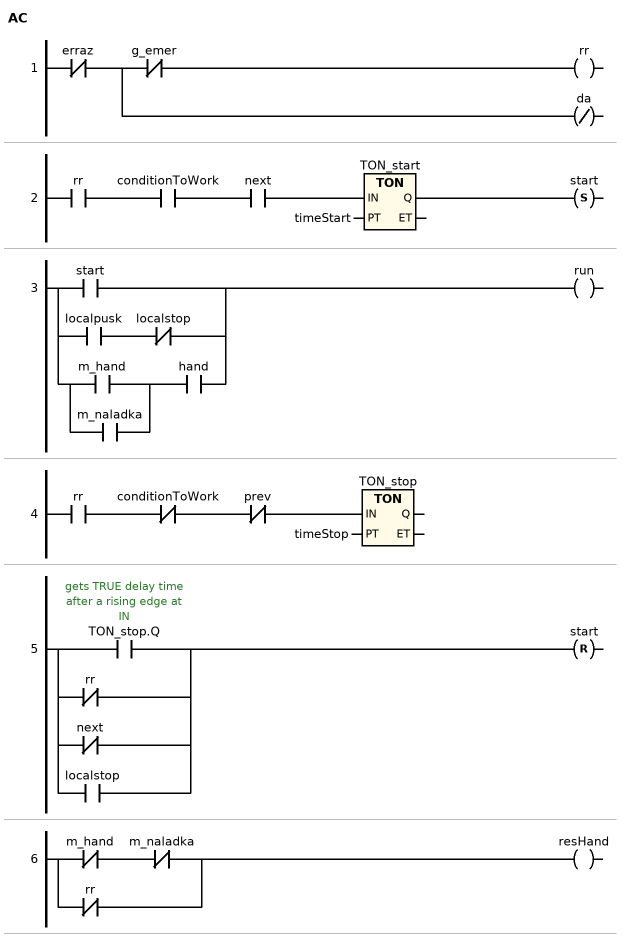
// NETWORK 1
_w1 := NOT erraz;
rr := _w1 AND NOT g_emer;
da := NOT _w1;

// NETWORK 2
TON_start(IN := rr AND conditionToWork AND next, PT := timeStart); // TON
start S= TON_start.Q;

// NETWORK 3
run := start OR localpusk AND NOT localstop OR (m_hand OR m_naladka) AND hand;

// NETWORK 4
TON_stop(IN := rr AND NOT conditionToWork AND NOT prev, PT := timeStop); // TON

// NETWORK 5
//   TON_stop.Q: gets TRUE delay time after a rising edge at IN
start R= TON_stop.Q OR NOT rr OR NOT next OR localstop;

// NETWORK 6
resHand := NOT m_hand AND NOT m_naladka OR NOT rr;

END_FUNCTION_BLOCK

// PLC_241/Application/FB/Noria/N
FUNCTION_BLOCK N
VAR_INPUT
	dks: BOOL;
	dsl1: BOOL;
	dsl2: BOOL;
	dp: BOOL;
	localpusk: BOOL;
	localstop: BOOL;
	erraz: BOOL;
	timeDKS: TIME;
	timeDSL: TIME;
	timeDP: TIME;
	timeStart: TIME;
	timeStop: TIME;
	next: BOOL;
	prev: BOOL;
	conditionToWork: BOOL;
	ressetErrors: BOOL;
	g_emer: BOOL;
	m_hand: BOOL;
	m_naladka: BOOL;
	hand: BOOL;
	offdks: BOOL;
	offdsl1: BOOL;
	offdsl2: BOOL;
	offdp: BOOL;
END_VAR
VAR_OUTPUT
	run: BOOL;
	rr: BOOL;
	da: BOOL;
	errDKS: BOOL;
	errDSL1: BOOL;
	errDSL2: BOOL;
	errDP: BOOL;
	resHand: BOOL;
END_VAR
VAR
	TON_DKS1: TON;
	TON_DKS2: TON;
	TON_DSL1: TON;
	TON_DSL2: TON;
	TON_DP: TON;
	TON_start: TON;
	start: BOOL;
	TON_stop: TON;
END_VAR
VAR // added by the converter: edge detectors and wires of the graphical bodies
    _w1 : BOOL;
END_VAR

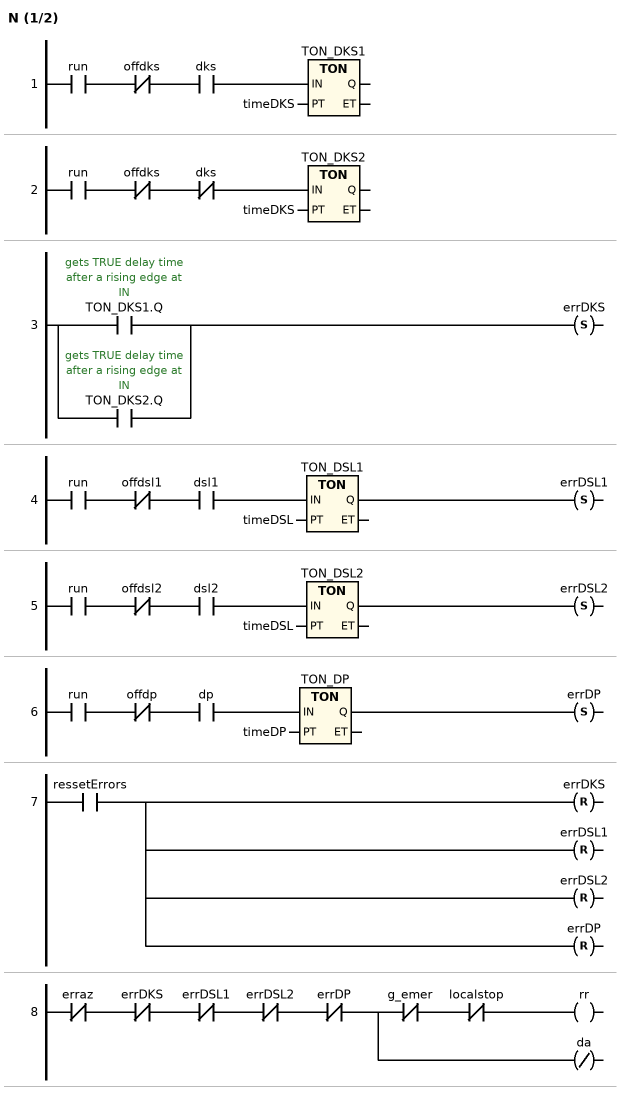
// NETWORK 1
TON_DKS1(IN := run AND NOT offdks AND dks, PT := timeDKS); // TON

// NETWORK 2
TON_DKS2(IN := run AND NOT offdks AND NOT dks, PT := timeDKS); // TON

// NETWORK 3
//   TON_DKS1.Q: gets TRUE delay time after a rising edge at IN
//   TON_DKS2.Q: gets TRUE delay time after a rising edge at IN
errDKS S= TON_DKS1.Q OR TON_DKS2.Q;

// NETWORK 4
TON_DSL1(IN := run AND NOT offdsl1 AND dsl1, PT := timeDSL); // TON
errDSL1 S= TON_DSL1.Q;

// NETWORK 5
TON_DSL2(IN := run AND NOT offdsl2 AND dsl2, PT := timeDSL); // TON
errDSL2 S= TON_DSL2.Q;

// NETWORK 6
TON_DP(IN := run AND NOT offdp AND dp, PT := timeDP); // TON
errDP S= TON_DP.Q;

// NETWORK 7
errDKS R= ressetErrors;
errDSL1 R= ressetErrors;
errDSL2 R= ressetErrors;
errDP R= ressetErrors;

// NETWORK 8
_w1 := NOT erraz AND NOT errDKS AND NOT errDSL1 AND NOT errDSL2 AND NOT errDP;
rr := _w1 AND NOT g_emer AND NOT localstop;
da := NOT _w1;

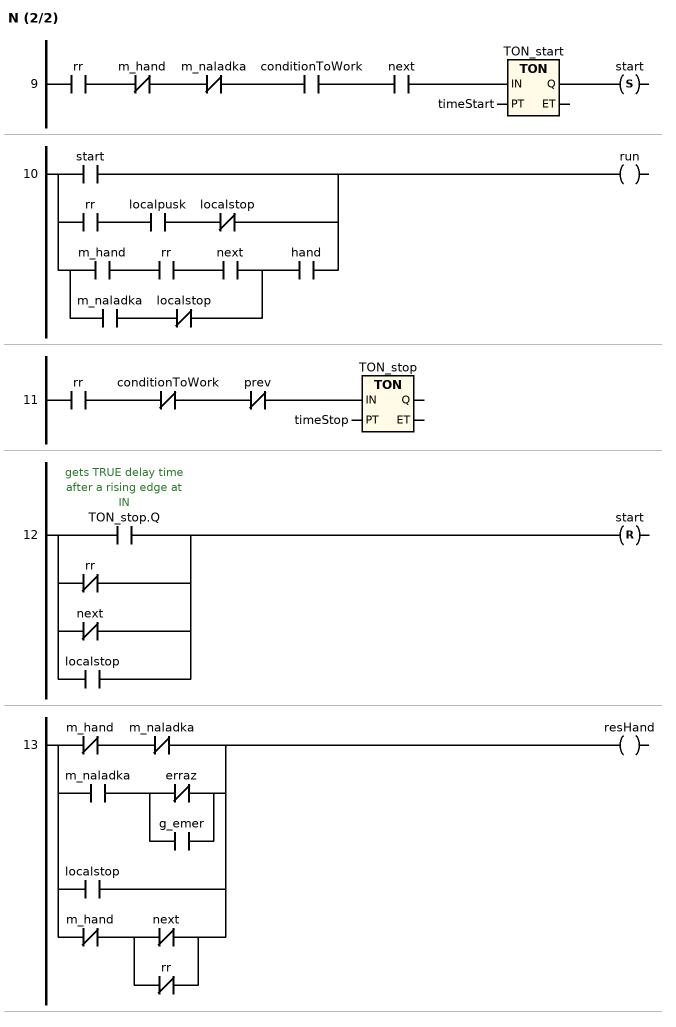
// NETWORK 9
TON_start(IN := rr AND NOT m_hand AND NOT m_naladka AND conditionToWork AND next, PT := timeStart); // TON
start S= TON_start.Q;

// NETWORK 10
run := start OR rr AND localpusk AND NOT localstop OR (m_hand AND rr AND next OR m_naladka AND NOT localstop) AND hand;

// NETWORK 11
TON_stop(IN := rr AND NOT conditionToWork AND NOT prev, PT := timeStop); // TON

// NETWORK 12
//   TON_stop.Q: gets TRUE delay time after a rising edge at IN
start R= TON_stop.Q OR NOT rr OR NOT next OR localstop;

// NETWORK 13
resHand := NOT m_hand AND NOT m_naladka OR m_naladka AND (NOT erraz OR g_emer) OR localstop OR NOT m_hand AND (NOT next OR NOT rr);

END_FUNCTION_BLOCK

// PLC_241/Application/FB/Flap/KP
FUNCTION_BLOCK KP
VAR_INPUT
	erraz: BOOL;
	pol_1: BOOL;
	pol_2: BOOL;
	conditionToWork_pol_1: BOOL;
	conditionToWork_pol_2: BOOL;
	timeLT: TIME;
	timePol_1: TIME;
	timePol_2: TIME;
	ressetErrors: BOOL;
	g_emer: BOOL;
	m_hand: BOOL;
	m_naladka: BOOL;
	hand_pol_1: BOOL;
	hand_pol_2: BOOL;
END_VAR
VAR_OUTPUT
	runPol_1: BOOL;
	runPol_2: BOOL;
	rr: BOOL;
	da: BOOL;
	errLT: BOOL;
	errConc: BOOL;
	stPol_1: BOOL;
	stPol_2: BOOL;
	resHand_pol_1: BOOL;
	resHand_pol_2: BOOL;
END_VAR
VAR
	TON_POL_1: TON;
	TON_LT: TON;
	TON_POL_2: TON;
END_VAR
VAR // added by the converter: edge detectors and wires of the graphical bodies
    _w1, _w2 : BOOL;
END_VAR

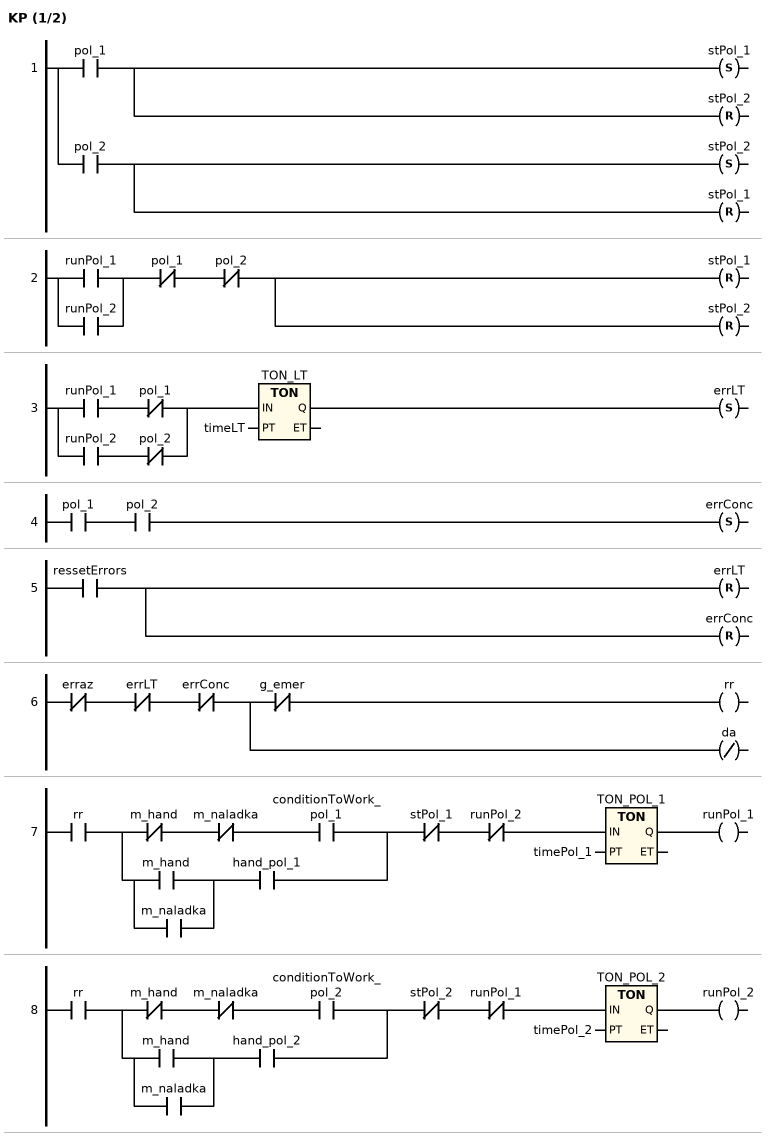
// NETWORK 1
stPol_1 S= pol_1;
stPol_2 R= pol_1;
stPol_2 S= pol_2;
stPol_1 R= pol_2;

// NETWORK 2
_w1 := (runPol_1 OR runPol_2) AND NOT pol_1 AND NOT pol_2;
stPol_1 R= _w1;
stPol_2 R= _w1;

// NETWORK 3
TON_LT(IN := runPol_1 AND NOT pol_1 OR runPol_2 AND NOT pol_2, PT := timeLT); // TON
errLT S= TON_LT.Q;

// NETWORK 4
errConc S= pol_1 AND pol_2;

// NETWORK 5
errLT R= ressetErrors;
errConc R= ressetErrors;

// NETWORK 6
_w2 := NOT erraz AND NOT errLT AND NOT errConc;
rr := _w2 AND NOT g_emer;
da := NOT _w2;

// NETWORK 7
TON_POL_1(IN := rr AND (NOT m_hand AND NOT m_naladka AND conditionToWork_pol_1 OR (m_hand OR m_naladka) AND hand_pol_1) AND NOT stPol_1 AND NOT runPol_2, PT := timePol_1); // TON
runPol_1 := TON_POL_1.Q;

// NETWORK 8
TON_POL_2(IN := rr AND (NOT m_hand AND NOT m_naladka AND conditionToWork_pol_2 OR (m_hand OR m_naladka) AND hand_pol_2) AND NOT stPol_2 AND NOT runPol_1, PT := timePol_2); // TON
runPol_2 := TON_POL_2.Q;

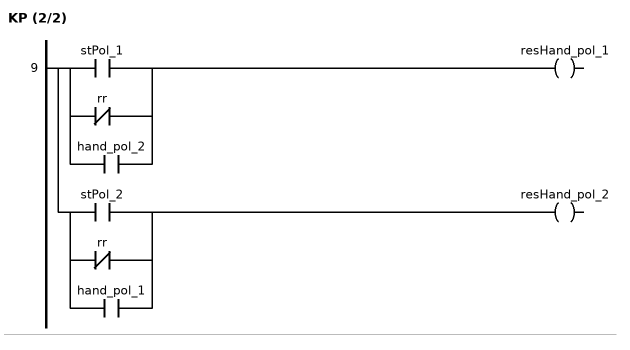
// NETWORK 9
resHand_pol_1 := stPol_1 OR NOT rr OR hand_pol_2;
resHand_pol_2 := stPol_2 OR NOT rr OR hand_pol_1;

END_FUNCTION_BLOCK

// PLC_241/Application/FB/scalperator/SCLP
FUNCTION_BLOCK SCLP
VAR_INPUT
	errpch: BOOL;
	prev: BOOL;
	next: BOOL;
	conditionToWork: BOOL;
	timeStart: TIME;
	timeStop: TIME;
	ressetErrors: BOOL;
	g_emer: BOOL;
	m_hand: BOOL;
	m_naladka: BOOL;
	hand: BOOL;
	
END_VAR
VAR_OUTPUT
	runPuskatel: BOOL;
	runPCH: BOOL;
	runRessetPCH: BOOL;
	rr: BOOL;
	da: BOOL;
	resHand: BOOL;
END_VAR
VAR
	TON_Start: TON;
	start: BOOL;
	TON_Stop: TON;
	TON_PCH_ON: TON;
END_VAR
VAR // added by the converter: edge detectors and wires of the graphical bodies
    _w1 : BOOL;
END_VAR

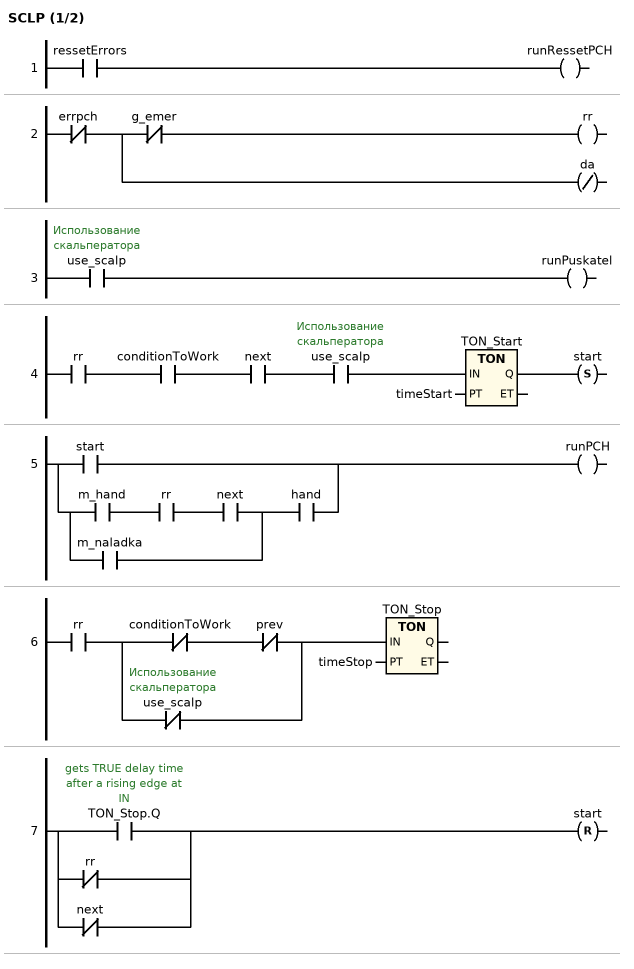
// NETWORK 1
runRessetPCH := ressetErrors;

// NETWORK 2
_w1 := NOT errpch;
rr := _w1 AND NOT g_emer;
da := NOT _w1;

// NETWORK 3
//   use_scalp: Использование скальператора
runPuskatel := use_scalp;

// NETWORK 4
//   use_scalp: Использование скальператора
TON_Start(IN := rr AND conditionToWork AND next AND use_scalp, PT := timeStart); // TON
start S= TON_Start.Q;

// NETWORK 5
runPCH := start OR (m_hand AND rr AND next OR m_naladka) AND hand;

// NETWORK 6
//   use_scalp: Использование скальператора
TON_Stop(IN := rr AND (NOT conditionToWork AND NOT prev OR NOT use_scalp), PT := timeStop); // TON

// NETWORK 7
//   TON_Stop.Q: gets TRUE delay time after a rising edge at IN
start R= TON_Stop.Q OR NOT rr OR NOT next;

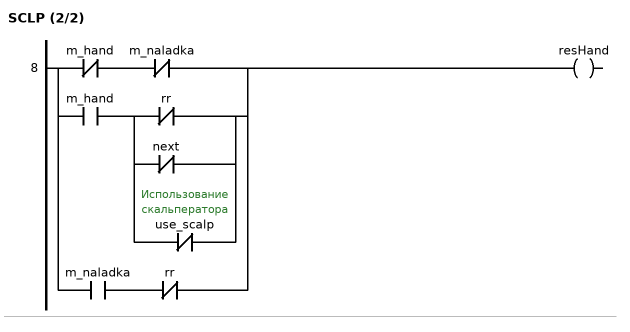
// NETWORK 8
//   use_scalp: Использование скальператора
resHand := NOT m_hand AND NOT m_naladka OR m_hand AND (NOT rr OR NOT next OR NOT use_scalp) OR m_naladka AND NOT rr;

END_FUNCTION_BLOCK

// PLC_241/Application/FB/SH/Z
FUNCTION_BLOCK Z
VAR_INPUT
	erraz: BOOL;
	opened: BOOL;
	closed: BOOL;
	next: BOOL;
	prev: BOOL;
	conditionToWork: BOOL;
	timeLT: TIME;
	timeOpen: TIME;
	timeClose: TIME;
	g_emer: BOOL;
	ressetErrors: BOOL;
	m_hand: BOOL;
	m_naladka: BOOL;
	hand_open: BOOL;
	hand_close: BOOL;
END_VAR
VAR_OUTPUT
	runOpen: BOOL; 
	runClose: BOOL;
	rr: BOOL;
	da: BOOL;
	errLT: BOOL;
	errConc: BOOL;
	resHand_open: BOOL;
	resHand_close: BOOL;
END_VAR
VAR
	TON_LT: TON;
	TON_open: TON;
	TON_close: TON;
END_VAR
VAR // added by the converter: edge detectors and wires of the graphical bodies
    _w1 : BOOL;
END_VAR

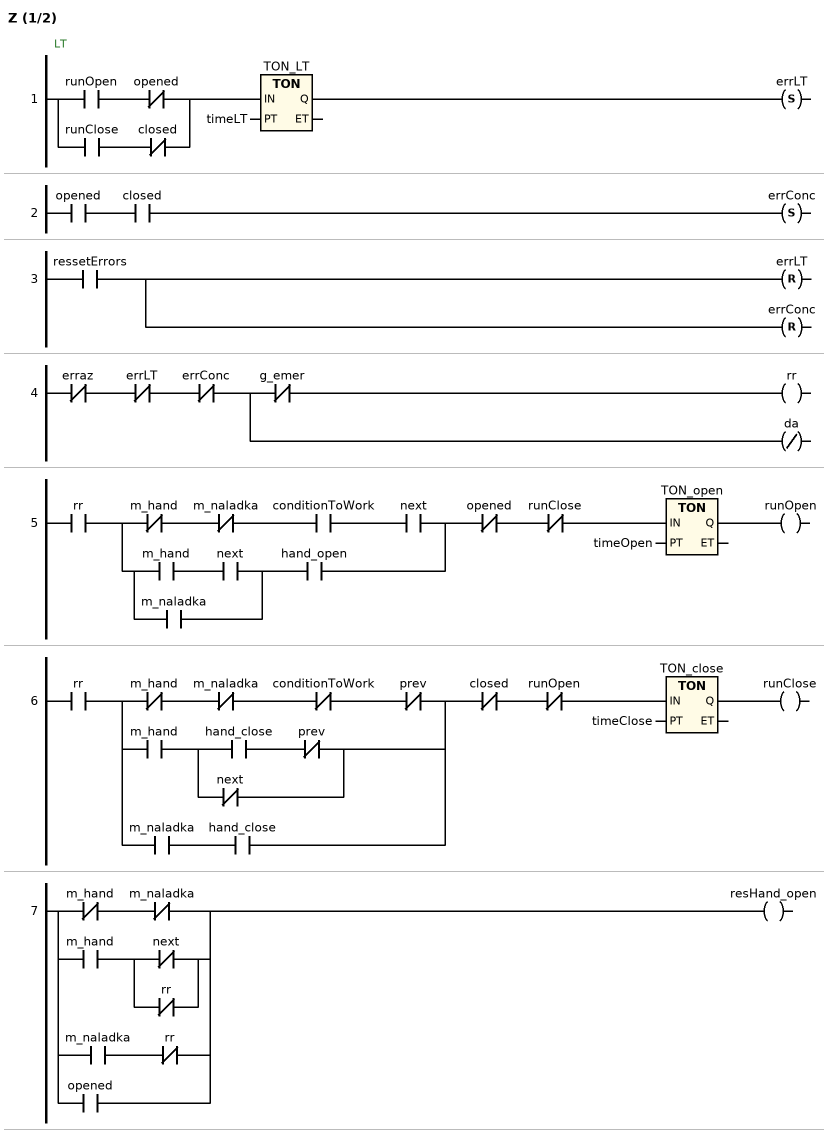
// NETWORK 1
// LT
TON_LT(IN := runOpen AND NOT opened OR runClose AND NOT closed, PT := timeLT); // TON
errLT S= TON_LT.Q;

// NETWORK 2
errConc S= opened AND closed;

// NETWORK 3
errLT R= ressetErrors;
errConc R= ressetErrors;

// NETWORK 4
_w1 := NOT erraz AND NOT errLT AND NOT errConc;
rr := _w1 AND NOT g_emer;
da := NOT _w1;

// NETWORK 5
TON_open(IN := rr AND (NOT m_hand AND NOT m_naladka AND conditionToWork AND next OR (m_hand AND next OR m_naladka) AND hand_open) AND NOT opened AND NOT runClose, PT := timeOpen); // TON
runOpen := TON_open.Q;

// NETWORK 6
TON_close(IN := rr AND (NOT m_hand AND NOT m_naladka AND NOT conditionToWork AND NOT prev OR m_hand AND (hand_close AND NOT prev OR NOT next) OR m_naladka AND hand_close) AND NOT closed AND NOT runOpen, PT := timeClose); // TON
runClose := TON_close.Q;

// NETWORK 7
resHand_open := NOT m_hand AND NOT m_naladka OR m_hand AND (NOT next OR NOT rr) OR m_naladka AND NOT rr OR opened;

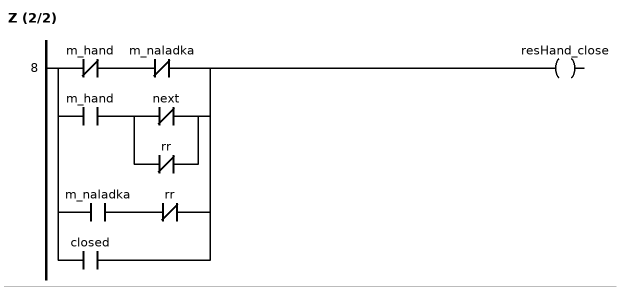
// NETWORK 8
resHand_close := NOT m_hand AND NOT m_naladka OR m_hand AND (NOT next OR NOT rr) OR m_naladka AND NOT rr OR closed;

END_FUNCTION_BLOCK

// PLC_241/Application/POU/prgLoad_K
PROGRAM prgLoad_K
VAR
	N_21200: N;
	Step_K: INT;
	imp_K: BOOL;
	imp_dvy_201: BOOL;
	imp_dvy_202: BOOL;
	imp_dvy_203: BOOL;
	imp_dvy_204: BOOL;
	TON_imp_bunk_201: TON;
	pause_load_K: BOOL;
	TON_imp_bunk_202: TON;
	TON_imp_bunk_203: TON;
	TON_imp_bunk_204: TON;
	TON_pause_K: TON;
	Shnek_21300: Shnek;
	TOF_next_shnek_21300: TOF;
	TP_STEP_K: TP;
	Z_21310: Z;
	Z_21320: Z;
	Z_21330: Z;
	check_K: BOOL;
	imp_nextBunk_K: BOOL;
	TON_Resset_modeLoad_k: TON;
END_VAR
VAR // added by the converter: edge detectors and wires of the graphical bodies
    _rt1, _rt2, _rt3, _rt4, _rt5, _rt6, _rt7, _rt8, _rt9, _rt10, _rt11, _rt12, _rt13 : R_TRIG;
    _w1, _w2, _w3, _w4, _w5, _w6 : BOOL;
END_VAR

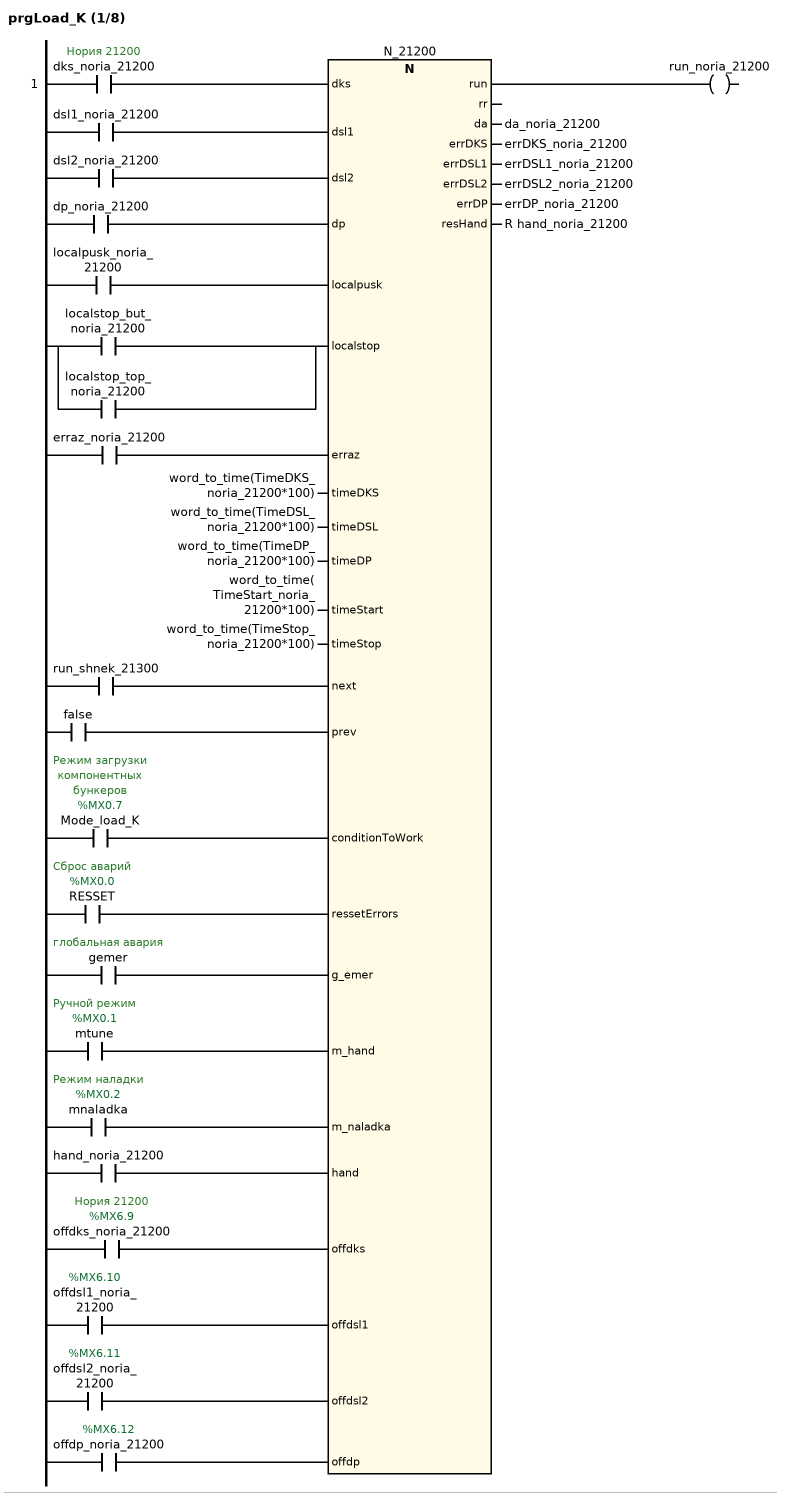
// NETWORK 1
//   dks_noria_21200: Нория 21200
//   Mode_load_K: Режим загрузки компонентных бункеров | AT %MX0.7
//   RESSET: Сброс аварий | AT %MX0.0
//   gemer: глобальная авария
//   mtune: Ручной режим | AT %MX0.1
//   mnaladka: Режим наладки | AT %MX0.2
//   offdks_noria_21200: Нория 21200 | AT %MX6.9
//   offdsl1_noria_21200: AT %MX6.10
//   offdsl2_noria_21200: AT %MX6.11
//   offdp_noria_21200: AT %MX6.12
//   errDKS_noria_21200: Нория 21200
N_21200(
    dks := dks_noria_21200,
    dsl1 := dsl1_noria_21200,
    dsl2 := dsl2_noria_21200,
    dp := dp_noria_21200,
    localpusk := localpusk_noria_21200,
    localstop := localstop_but_noria_21200 OR localstop_top_noria_21200,
    erraz := erraz_noria_21200,
    timeDKS := word_to_time(TimeDKS_noria_21200*100),
    timeDSL := word_to_time(TimeDSL_noria_21200*100),
    timeDP := word_to_time(TimeDP_noria_21200*100),
    timeStart := word_to_time(TimeStart_noria_21200*100),
    timeStop := word_to_time(TimeStop_noria_21200*100),
    next := run_shnek_21300,
    prev := false,
    conditionToWork := Mode_load_K,
    ressetErrors := RESSET,
    g_emer := gemer,
    m_hand := mtune,
    m_naladka := mnaladka,
    hand := hand_noria_21200,
    offdks := offdks_noria_21200,
    offdsl1 := offdsl1_noria_21200,
    offdsl2 := offdsl2_noria_21200,
    offdp := offdp_noria_21200,
    da => da_noria_21200,
    errDKS => errDKS_noria_21200,
    errDSL1 => errDSL1_noria_21200,
    errDSL2 => errDSL2_noria_21200,
    errDP => errDP_noria_21200); // N
hand_noria_21200 R= N_21200.resHand;
run_noria_21200 := N_21200.run;

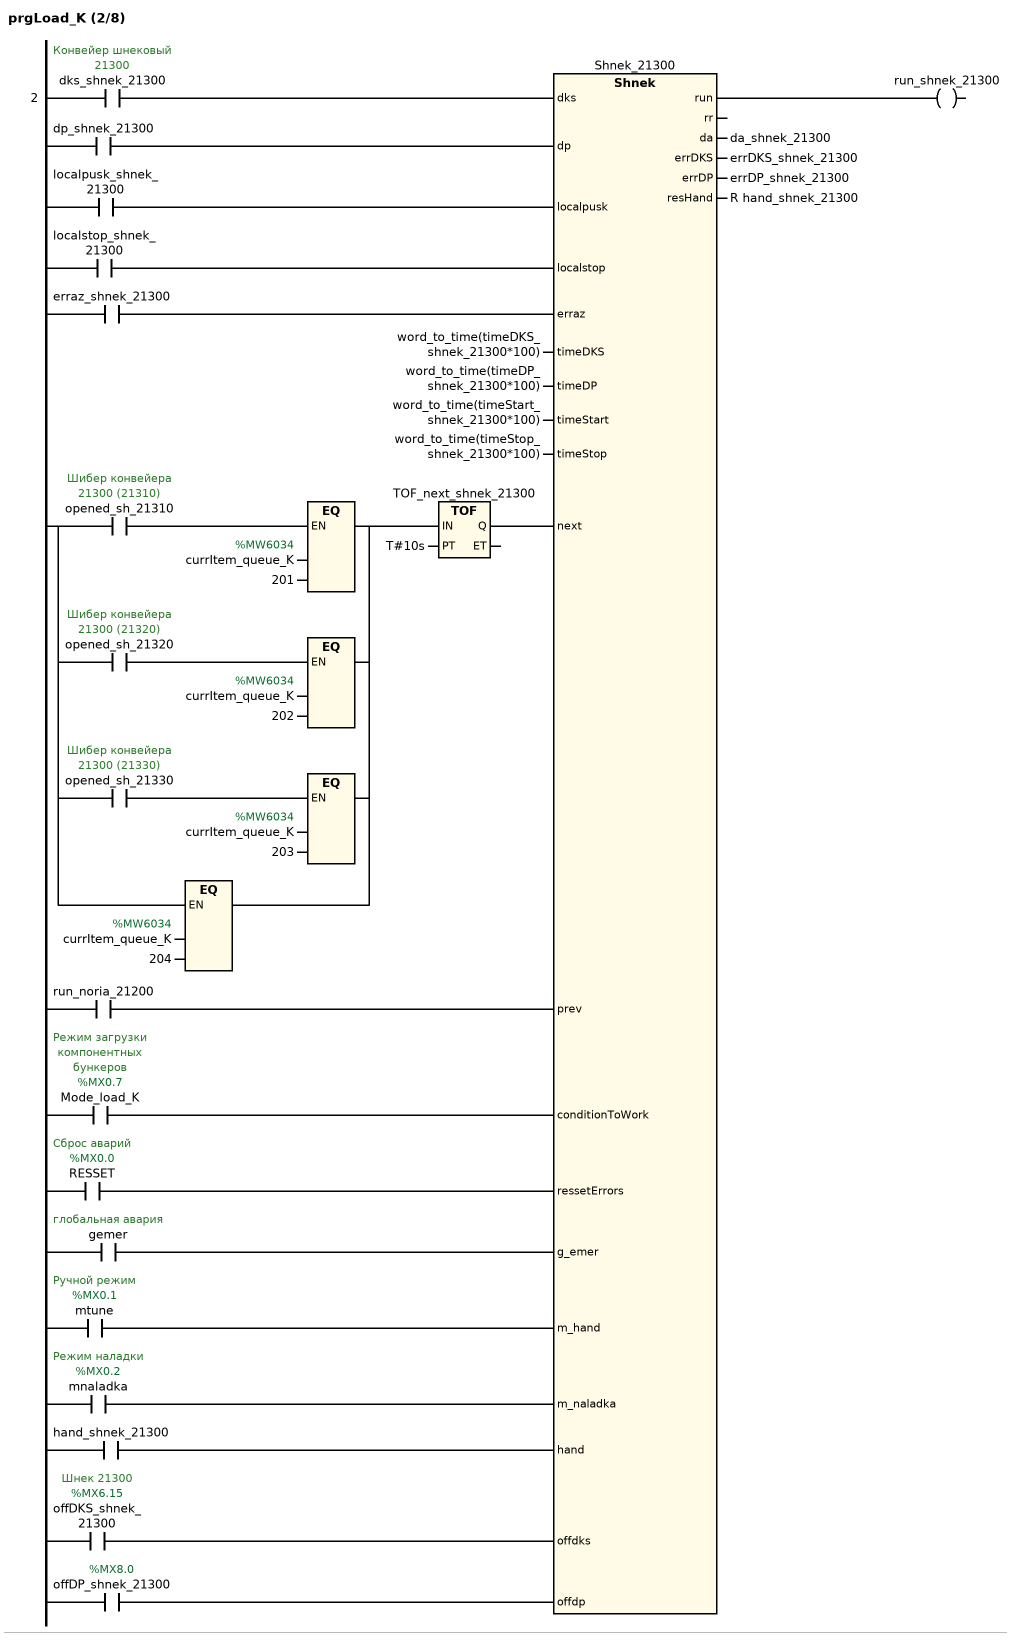
// NETWORK 2
//   dks_shnek_21300: Конвейер шнековый 21300
//   opened_sh_21310: Шибер конвейера 21300 (21310)
//   currItem_queue_K: Текущий бункер для загрузки в очереди компонентов | AT %MW6034
//   opened_sh_21320: Шибер конвейера 21300 (21320)
//   opened_sh_21330: Шибер конвейера 21300 (21330)
//   Mode_load_K: Режим загрузки компонентных бункеров | AT %MX0.7
//   RESSET: Сброс аварий | AT %MX0.0
//   gemer: глобальная авария
//   mtune: Ручной режим | AT %MX0.1
//   mnaladka: Режим наладки | AT %MX0.2
//   offDKS_shnek_21300: Шнек 21300 | AT %MX6.15
//   offDP_shnek_21300: AT %MX8.0
//   errDKS_shnek_21300: Шнек 21300
TOF_next_shnek_21300(IN := opened_sh_21310 AND currItem_queue_K = 201 OR opened_sh_21320 AND currItem_queue_K = 202 OR opened_sh_21330 AND currItem_queue_K = 203 OR currItem_queue_K = 204, PT := T#10s); // TOF
Shnek_21300(
    dks := dks_shnek_21300,
    dp := dp_shnek_21300,
    localpusk := localpusk_shnek_21300,
    localstop := localstop_shnek_21300,
    erraz := erraz_shnek_21300,
    timeDKS := word_to_time(timeDKS_shnek_21300*100),
    timeDP := word_to_time(timeDP_shnek_21300*100),
    timeStart := word_to_time(timeStart_shnek_21300*100),
    timeStop := word_to_time(timeStop_shnek_21300*100),
    next := TOF_next_shnek_21300.Q,
    prev := run_noria_21200,
    conditionToWork := Mode_load_K,
    ressetErrors := RESSET,
    g_emer := gemer,
    m_hand := mtune,
    m_naladka := mnaladka,
    hand := hand_shnek_21300,
    offdks := offDKS_shnek_21300,
    offdp := offDP_shnek_21300,
    da => da_shnek_21300,
    errDKS => errDKS_shnek_21300,
    errDP => errDP_shnek_21300); // Shnek
hand_shnek_21300 R= Shnek_21300.resHand;
run_shnek_21300 := Shnek_21300.run;

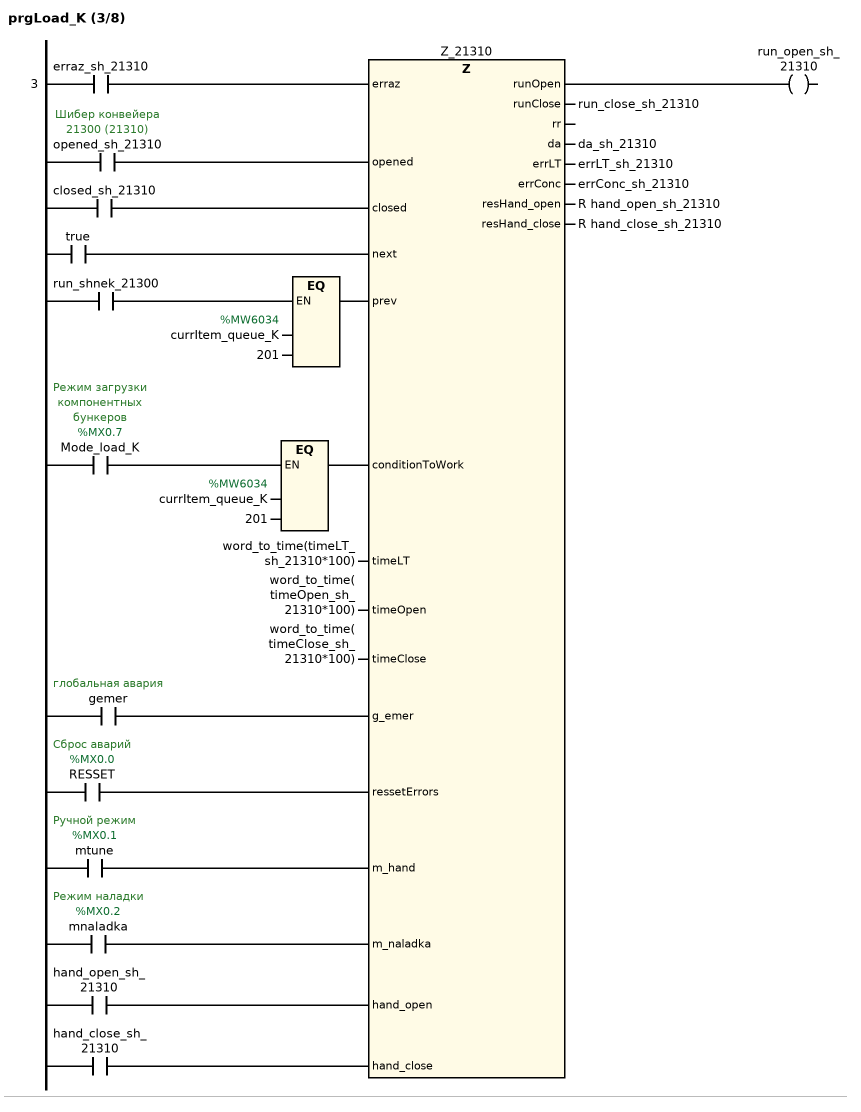
// NETWORK 3
//   opened_sh_21310: Шибер конвейера 21300 (21310)
//   currItem_queue_K: Текущий бункер для загрузки в очереди компонентов | AT %MW6034
//   Mode_load_K: Режим загрузки компонентных бункеров | AT %MX0.7
//   gemer: глобальная авария
//   RESSET: Сброс аварий | AT %MX0.0
//   mtune: Ручной режим | AT %MX0.1
//   mnaladka: Режим наладки | AT %MX0.2
//   errLT_sh_21310: Шибер 21310
Z_21310(
    erraz := erraz_sh_21310,
    opened := opened_sh_21310,
    closed := closed_sh_21310,
    next := true,
    prev := run_shnek_21300 AND currItem_queue_K = 201,
    conditionToWork := Mode_load_K AND currItem_queue_K = 201,
    timeLT := word_to_time(timeLT_sh_21310*100),
    timeOpen := word_to_time(timeOpen_sh_21310*100),
    timeClose := word_to_time(timeClose_sh_21310*100),
    g_emer := gemer,
    ressetErrors := RESSET,
    m_hand := mtune,
    m_naladka := mnaladka,
    hand_open := hand_open_sh_21310,
    hand_close := hand_close_sh_21310,
    runClose => run_close_sh_21310,
    da => da_sh_21310,
    errLT => errLT_sh_21310,
    errConc => errConc_sh_21310); // Z
hand_open_sh_21310 R= Z_21310.resHand_open;
hand_close_sh_21310 R= Z_21310.resHand_close;
run_open_sh_21310 := Z_21310.runOpen;

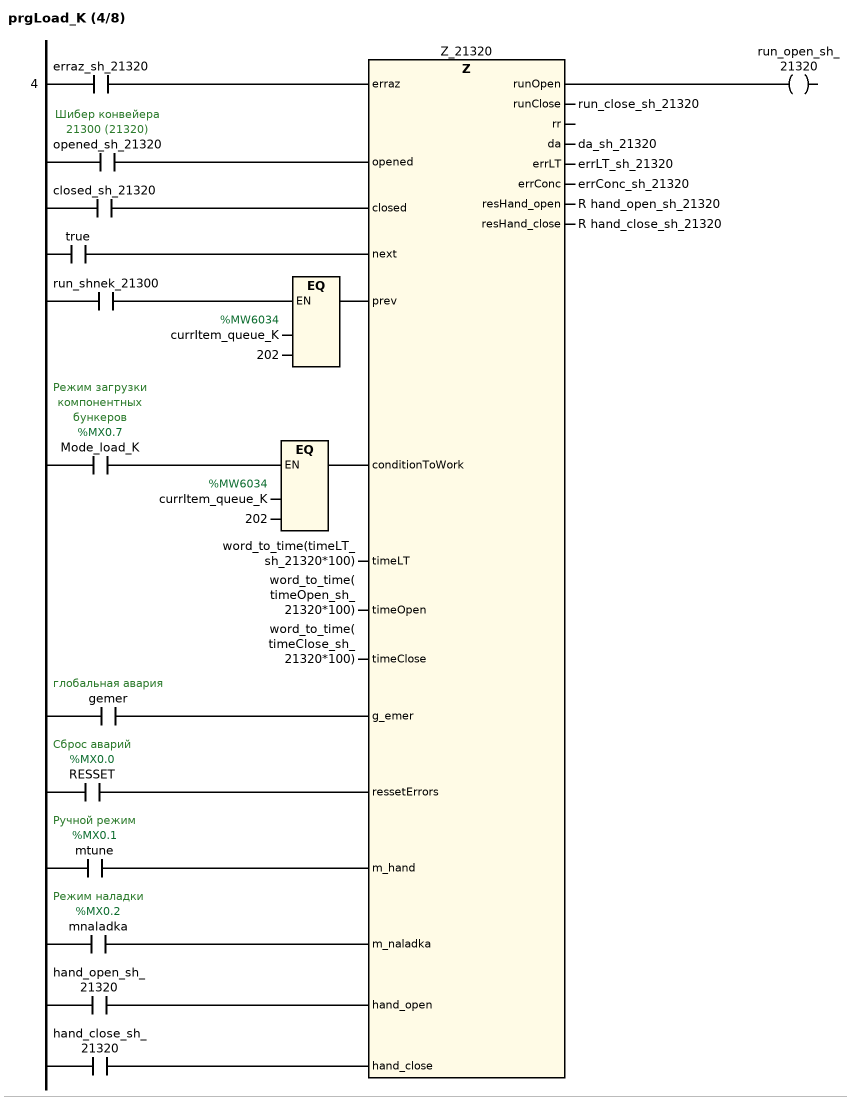
// NETWORK 4
//   opened_sh_21320: Шибер конвейера 21300 (21320)
//   currItem_queue_K: Текущий бункер для загрузки в очереди компонентов | AT %MW6034
//   Mode_load_K: Режим загрузки компонентных бункеров | AT %MX0.7
//   gemer: глобальная авария
//   RESSET: Сброс аварий | AT %MX0.0
//   mtune: Ручной режим | AT %MX0.1
//   mnaladka: Режим наладки | AT %MX0.2
//   errLT_sh_21320: Шибер 21320
Z_21320(
    erraz := erraz_sh_21320,
    opened := opened_sh_21320,
    closed := closed_sh_21320,
    next := true,
    prev := run_shnek_21300 AND currItem_queue_K = 202,
    conditionToWork := Mode_load_K AND currItem_queue_K = 202,
    timeLT := word_to_time(timeLT_sh_21320*100),
    timeOpen := word_to_time(timeOpen_sh_21320*100),
    timeClose := word_to_time(timeClose_sh_21320*100),
    g_emer := gemer,
    ressetErrors := RESSET,
    m_hand := mtune,
    m_naladka := mnaladka,
    hand_open := hand_open_sh_21320,
    hand_close := hand_close_sh_21320,
    runClose => run_close_sh_21320,
    da => da_sh_21320,
    errLT => errLT_sh_21320,
    errConc => errConc_sh_21320); // Z
hand_open_sh_21320 R= Z_21320.resHand_open;
hand_close_sh_21320 R= Z_21320.resHand_close;
run_open_sh_21320 := Z_21320.runOpen;

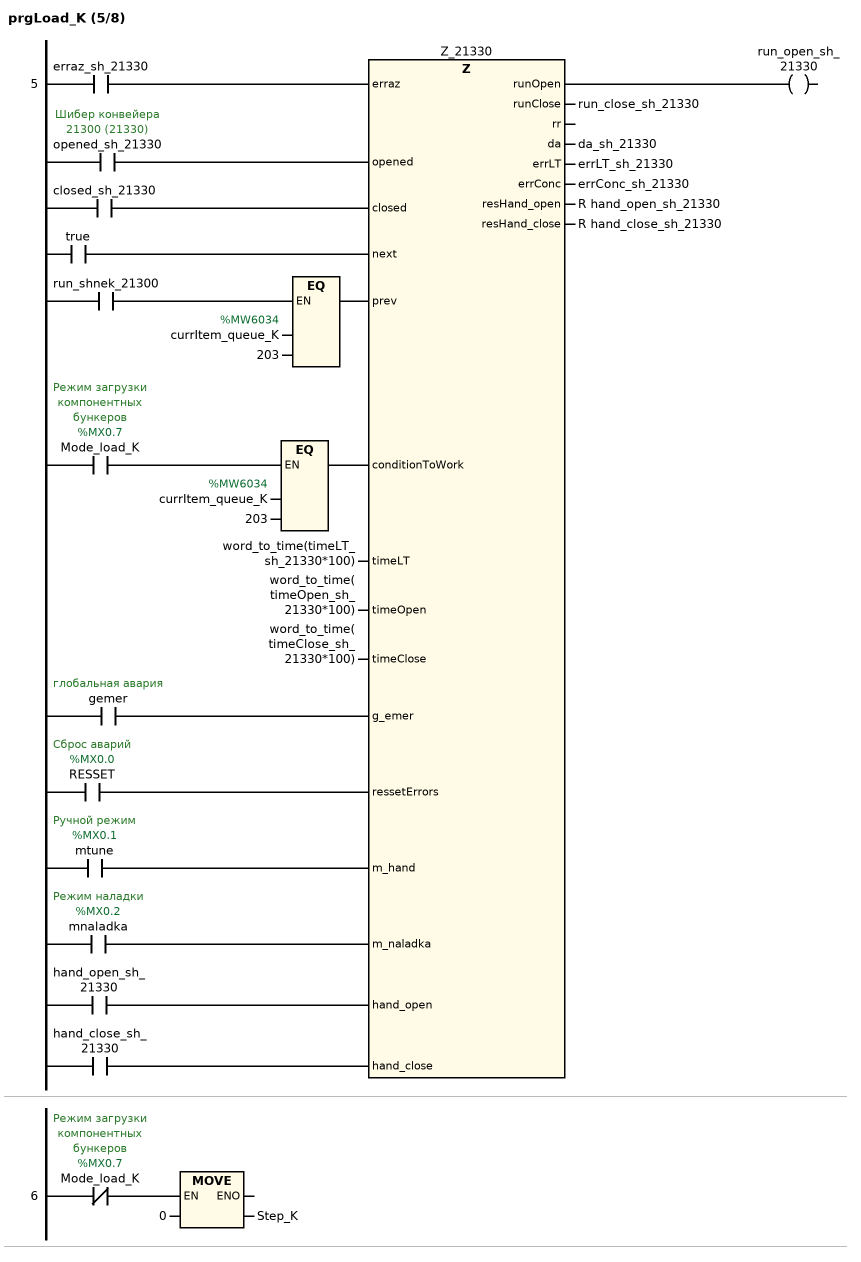
// NETWORK 5
//   opened_sh_21330: Шибер конвейера 21300 (21330)
//   currItem_queue_K: Текущий бункер для загрузки в очереди компонентов | AT %MW6034
//   Mode_load_K: Режим загрузки компонентных бункеров | AT %MX0.7
//   gemer: глобальная авария
//   RESSET: Сброс аварий | AT %MX0.0
//   mtune: Ручной режим | AT %MX0.1
//   mnaladka: Режим наладки | AT %MX0.2
//   errLT_sh_21330: Шибер 21330
Z_21330(
    erraz := erraz_sh_21330,
    opened := opened_sh_21330,
    closed := closed_sh_21330,
    next := true,
    prev := run_shnek_21300 AND currItem_queue_K = 203,
    conditionToWork := Mode_load_K AND currItem_queue_K = 203,
    timeLT := word_to_time(timeLT_sh_21330*100),
    timeOpen := word_to_time(timeOpen_sh_21330*100),
    timeClose := word_to_time(timeClose_sh_21330*100),
    g_emer := gemer,
    ressetErrors := RESSET,
    m_hand := mtune,
    m_naladka := mnaladka,
    hand_open := hand_open_sh_21330,
    hand_close := hand_close_sh_21330,
    runClose => run_close_sh_21330,
    da => da_sh_21330,
    errLT => errLT_sh_21330,
    errConc => errConc_sh_21330); // Z
hand_open_sh_21330 R= Z_21330.resHand_open;
hand_close_sh_21330 R= Z_21330.resHand_close;
run_open_sh_21330 := Z_21330.runOpen;

// NETWORK 6
//   Mode_load_K: Режим загрузки компонентных бункеров | AT %MX0.7
IF NOT Mode_load_K THEN Step_K := 0; END_IF

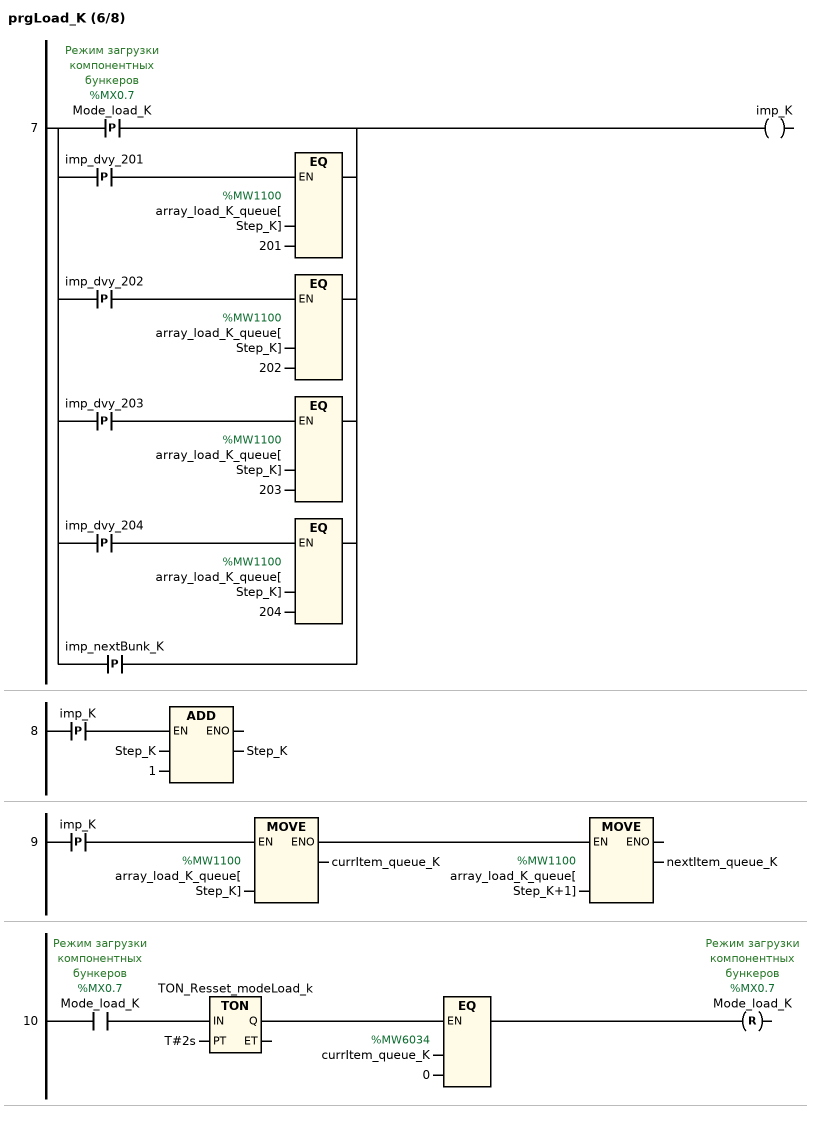
// NETWORK 7
//   Mode_load_K: Режим загрузки компонентных бункеров | AT %MX0.7
//   array_load_K_queue[Step_K]: Массив очереди загрузки компонентов | AT %MW1100
_rt1(CLK := Mode_load_K);
_rt2(CLK := imp_dvy_201);
_rt3(CLK := imp_dvy_202);
_rt4(CLK := imp_dvy_203);
_rt5(CLK := imp_dvy_204);
_rt6(CLK := imp_nextBunk_K);
imp_K := _rt1.Q OR _rt2.Q AND array_load_K_queue[Step_K] = 201 OR _rt3.Q AND array_load_K_queue[Step_K] = 202 OR _rt4.Q AND array_load_K_queue[Step_K] = 203 OR _rt5.Q AND array_load_K_queue[Step_K] = 204 OR _rt6.Q;

// NETWORK 8
_rt7(CLK := imp_K);
IF _rt7.Q THEN Step_K := Step_K + 1; END_IF

// NETWORK 9
//   array_load_K_queue[Step_K]: Массив очереди загрузки компонентов | AT %MW1100
//   currItem_queue_K: Текущий бункер для загрузки в очереди компонентов | AT %MW6034
//   array_load_K_queue[Step_K+1]: Массив очереди загрузки компонентов | AT %MW1100
//   nextItem_queue_K: Следующий бункер для загрузки в очереди компонентов | AT %MW6035
_rt8(CLK := imp_K);
_w1 := _rt8.Q;
IF _w1 THEN currItem_queue_K := array_load_K_queue[Step_K]; END_IF
IF _w1 THEN nextItem_queue_K := array_load_K_queue[Step_K+1]; END_IF

// NETWORK 10
//   Mode_load_K: Режим загрузки компонентных бункеров | AT %MX0.7
//   currItem_queue_K: Текущий бункер для загрузки в очереди компонентов | AT %MW6034
TON_Resset_modeLoad_k(IN := Mode_load_K, PT := T#2s); // TON
Mode_load_K R= TON_Resset_modeLoad_k.Q AND currItem_queue_K = 0;

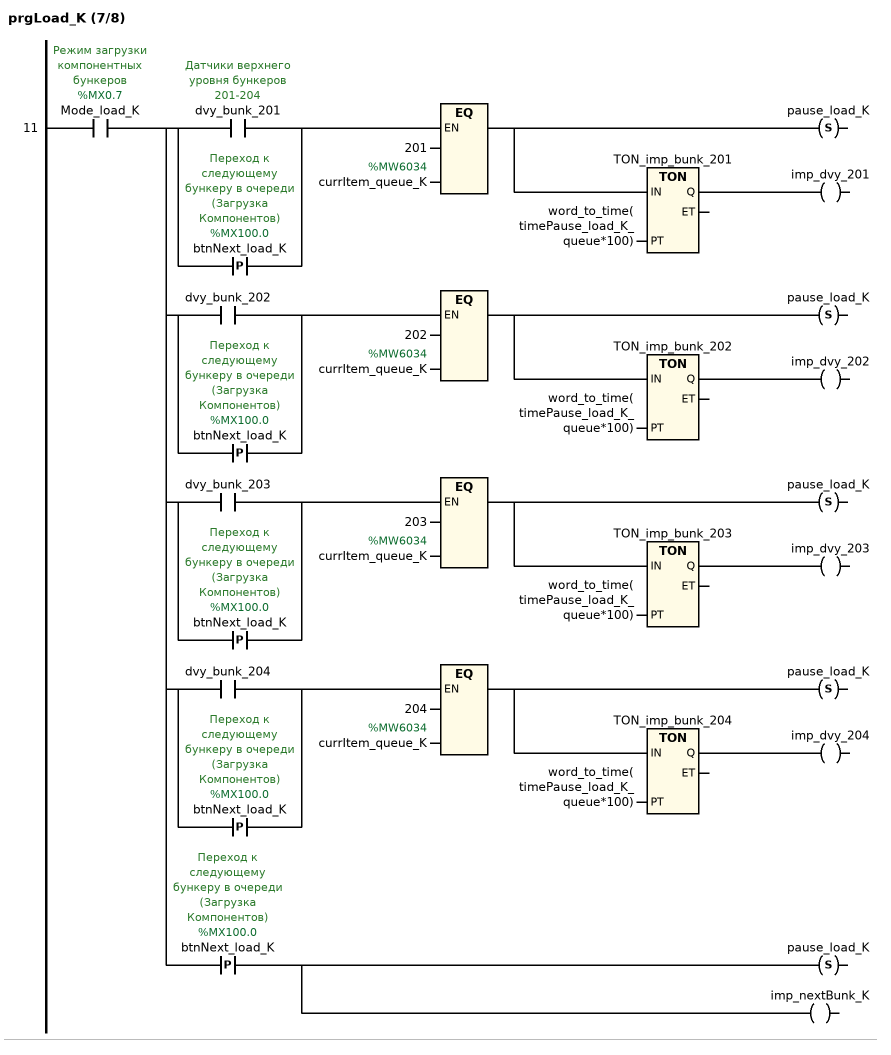
// NETWORK 11
//   Mode_load_K: Режим загрузки компонентных бункеров | AT %MX0.7
//   dvy_bunk_201: Датчики верхнего уровня бункеров 201-204
//   btnNext_load_K: Переход к следующему бункеру в очереди (Загрузка Компонентов) | AT %MX100.0
//   currItem_queue_K: Текущий бункер для загрузки в очереди компонентов | AT %MW6034
_rt9(CLK := btnNext_load_K);
_w2 := Mode_load_K AND (dvy_bunk_201 OR _rt9.Q) AND 201 = currItem_queue_K;
pause_load_K S= _w2;
TON_imp_bunk_201(IN := _w2, PT := word_to_time(timePause_load_K_queue*100)); // TON
imp_dvy_201 := TON_imp_bunk_201.Q;
_rt10(CLK := btnNext_load_K);
_w3 := Mode_load_K AND (dvy_bunk_202 OR _rt10.Q) AND 202 = currItem_queue_K;
pause_load_K S= _w3;
TON_imp_bunk_202(IN := _w3, PT := word_to_time(timePause_load_K_queue*100)); // TON
imp_dvy_202 := TON_imp_bunk_202.Q;
_rt11(CLK := btnNext_load_K);
_w4 := Mode_load_K AND (dvy_bunk_203 OR _rt11.Q) AND 203 = currItem_queue_K;
pause_load_K S= _w4;
TON_imp_bunk_203(IN := _w4, PT := word_to_time(timePause_load_K_queue*100)); // TON
imp_dvy_203 := TON_imp_bunk_203.Q;
_rt12(CLK := btnNext_load_K);
_w5 := Mode_load_K AND (dvy_bunk_204 OR _rt12.Q) AND 204 = currItem_queue_K;
pause_load_K S= _w5;
TON_imp_bunk_204(IN := _w5, PT := word_to_time(timePause_load_K_queue*100)); // TON
imp_dvy_204 := TON_imp_bunk_204.Q;
_rt13(CLK := btnNext_load_K);
_w6 := Mode_load_K AND _rt13.Q;
pause_load_K S= _w6;
imp_nextBunk_K := _w6;

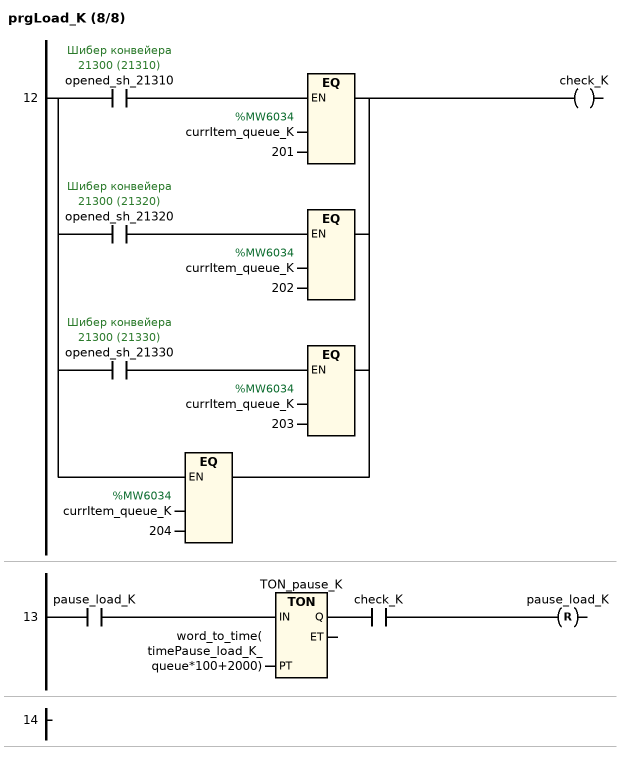
// NETWORK 12
//   opened_sh_21310: Шибер конвейера 21300 (21310)
//   currItem_queue_K: Текущий бункер для загрузки в очереди компонентов | AT %MW6034
//   opened_sh_21320: Шибер конвейера 21300 (21320)
//   opened_sh_21330: Шибер конвейера 21300 (21330)
check_K := opened_sh_21310 AND currItem_queue_K = 201 OR opened_sh_21320 AND currItem_queue_K = 202 OR opened_sh_21330 AND currItem_queue_K = 203 OR currItem_queue_K = 204;

// NETWORK 13
TON_pause_K(IN := pause_load_K, PT := word_to_time(timePause_load_K_queue*100+2000)); // TON
pause_load_K R= TON_pause_K.Q AND check_K;

// NETWORK 14

END_PROGRAM

// PLC_241/Application/FB/SKTR/Shnek
FUNCTION_BLOCK Shnek
VAR_INPUT
	dks: BOOL;
	dp: BOOL;
	localpusk: BOOL;
	localstop: BOOL;
	erraz: BOOL;
	timeDKS: TIME;
	timeDP: TIME;
	timeStart: TIME;
	timeStop: TIME;
	next: BOOL;
	prev: BOOL;
	conditionToWork: BOOL;
	ressetErrors: BOOL;
	g_emer: BOOL;
	m_hand: BOOL;
	m_naladka: BOOL;
	hand: BOOL;
	offdks: BOOL;
	offdp: BOOL;
	
END_VAR
VAR_OUTPUT
	run: BOOL;
	rr: BOOL;
	da: BOOL;
	errDKS: BOOL;
	errDP: BOOL;
	resHand: BOOL;
END_VAR
VAR
	TON_DKS_ON: TON;
	TON_DKS_OFF: TON;
	TON_DP: TON;
	TON_start: TON;
	start: BOOL;
	TON_Stop: TON;
END_VAR
VAR // added by the converter: edge detectors and wires of the graphical bodies
    _w1 : BOOL;
END_VAR

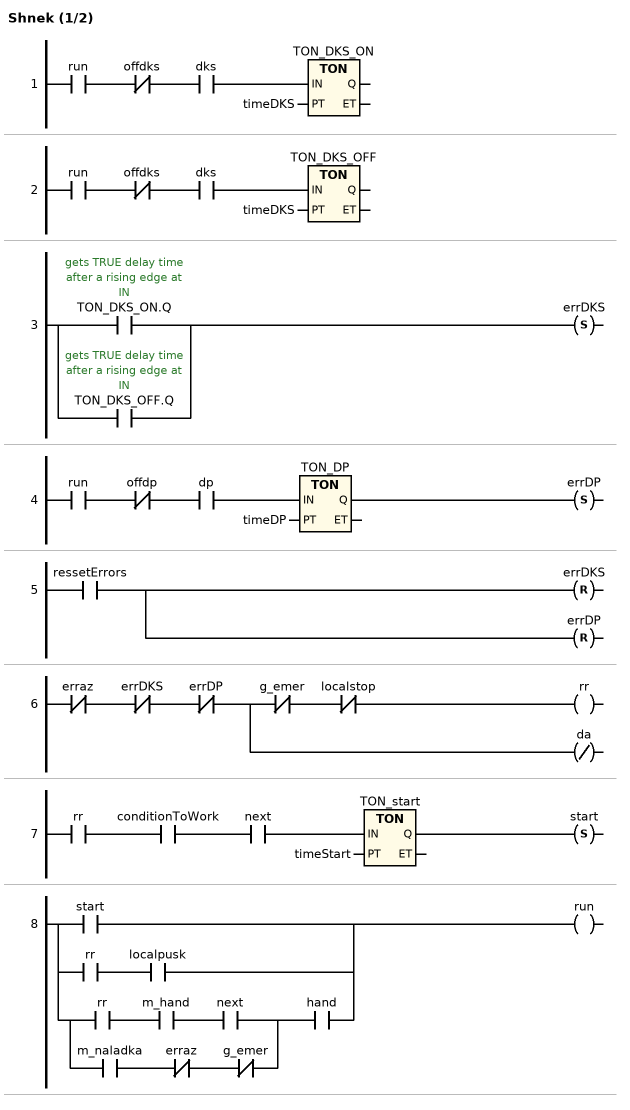
// NETWORK 1
TON_DKS_ON(IN := run AND NOT offdks AND dks, PT := timeDKS); // TON

// NETWORK 2
TON_DKS_OFF(IN := run AND NOT offdks AND dks, PT := timeDKS); // TON

// NETWORK 3
//   TON_DKS_ON.Q: gets TRUE delay time after a rising edge at IN
//   TON_DKS_OFF.Q: gets TRUE delay time after a rising edge at IN
errDKS S= TON_DKS_ON.Q OR TON_DKS_OFF.Q;

// NETWORK 4
TON_DP(IN := run AND NOT offdp AND dp, PT := timeDP); // TON
errDP S= TON_DP.Q;

// NETWORK 5
errDKS R= ressetErrors;
errDP R= ressetErrors;

// NETWORK 6
_w1 := NOT erraz AND NOT errDKS AND NOT errDP;
rr := _w1 AND NOT g_emer AND NOT localstop;
da := NOT _w1;

// NETWORK 7
TON_start(IN := rr AND conditionToWork AND next, PT := timeStart); // TON
start S= TON_start.Q;

// NETWORK 8
run := start OR rr AND localpusk OR (rr AND m_hand AND next OR m_naladka AND NOT erraz AND NOT g_emer) AND hand;

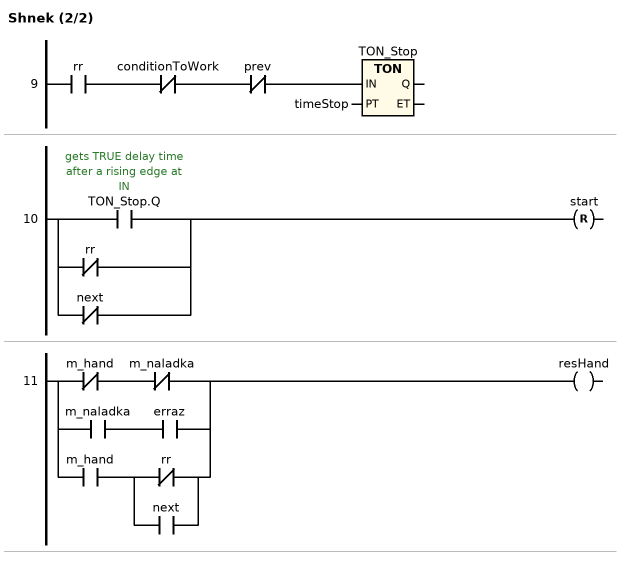
// NETWORK 9
TON_Stop(IN := rr AND NOT conditionToWork AND NOT prev, PT := timeStop); // TON

// NETWORK 10
//   TON_Stop.Q: gets TRUE delay time after a rising edge at IN
start R= TON_Stop.Q OR NOT rr OR NOT next;

// NETWORK 11
resHand := NOT m_hand AND NOT m_naladka OR m_naladka AND erraz OR m_hand AND (NOT rr OR next);

END_FUNCTION_BLOCK

// PLC_241/Application/POU/prgAdd_weight
PROGRAM prgAdd_weight
VAR
END_VAR
VAR // added by the converter: edge detectors and wires of the graphical bodies
    _w1, _w2 : BOOL;
END_VAR

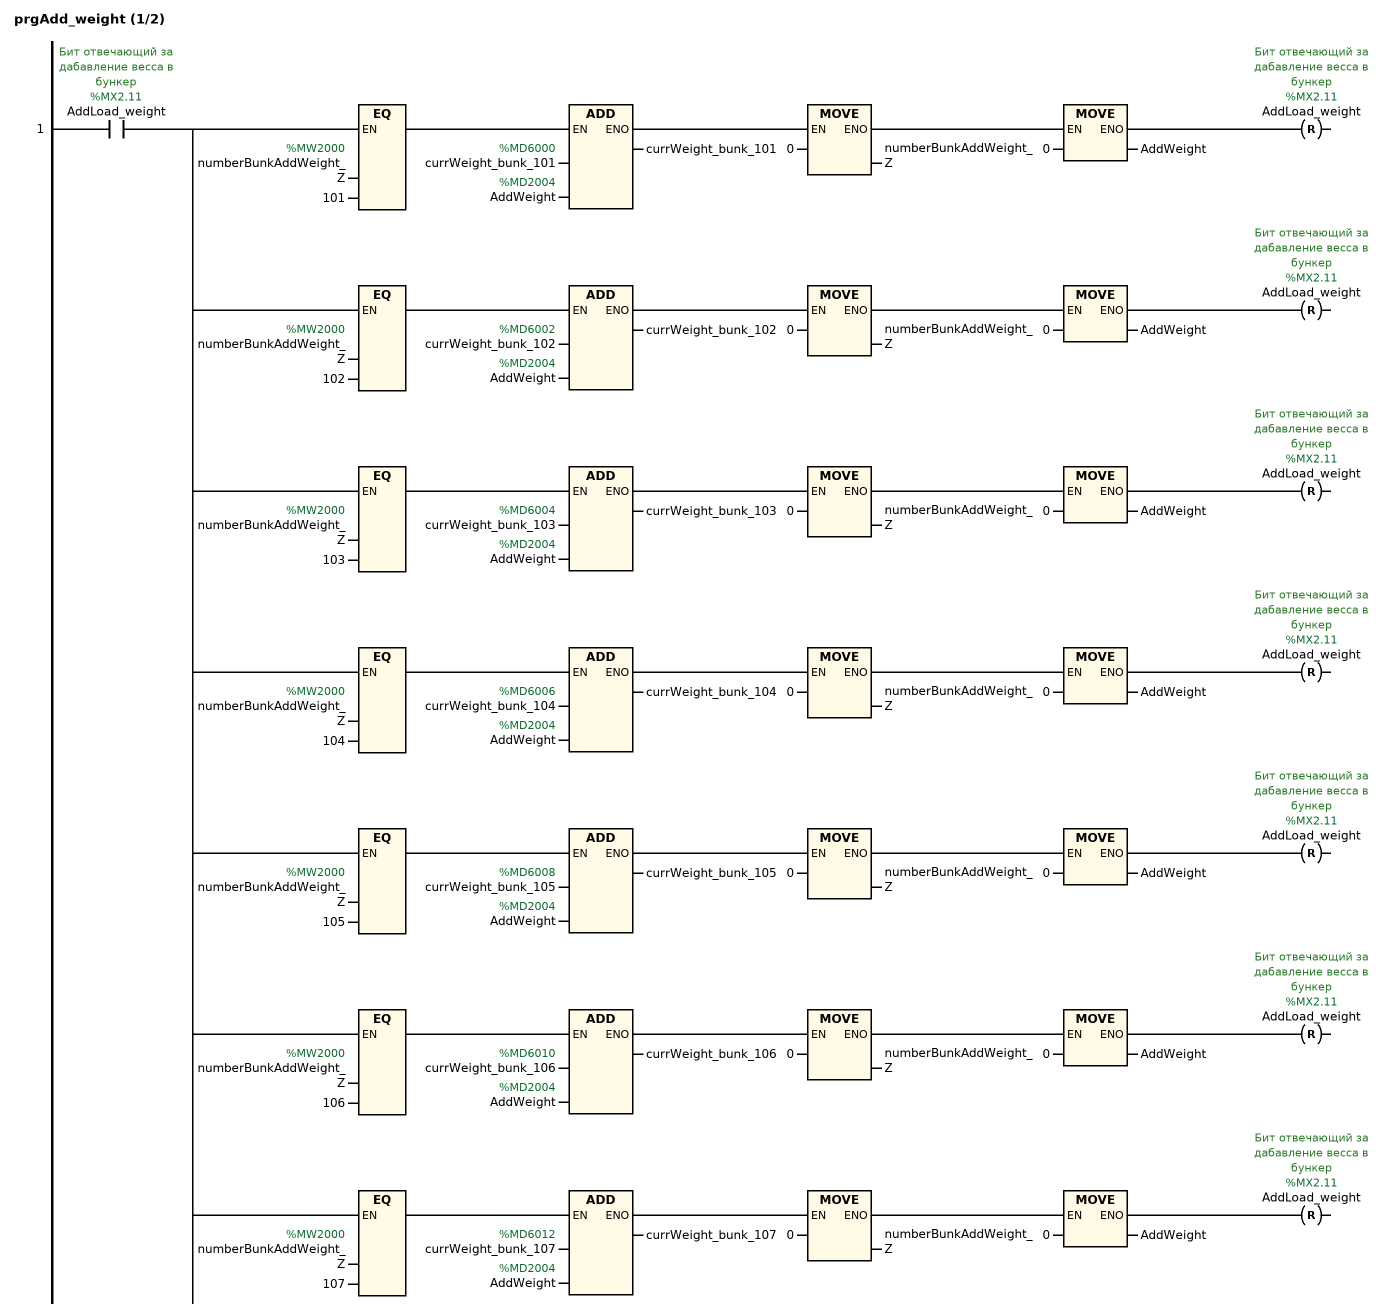
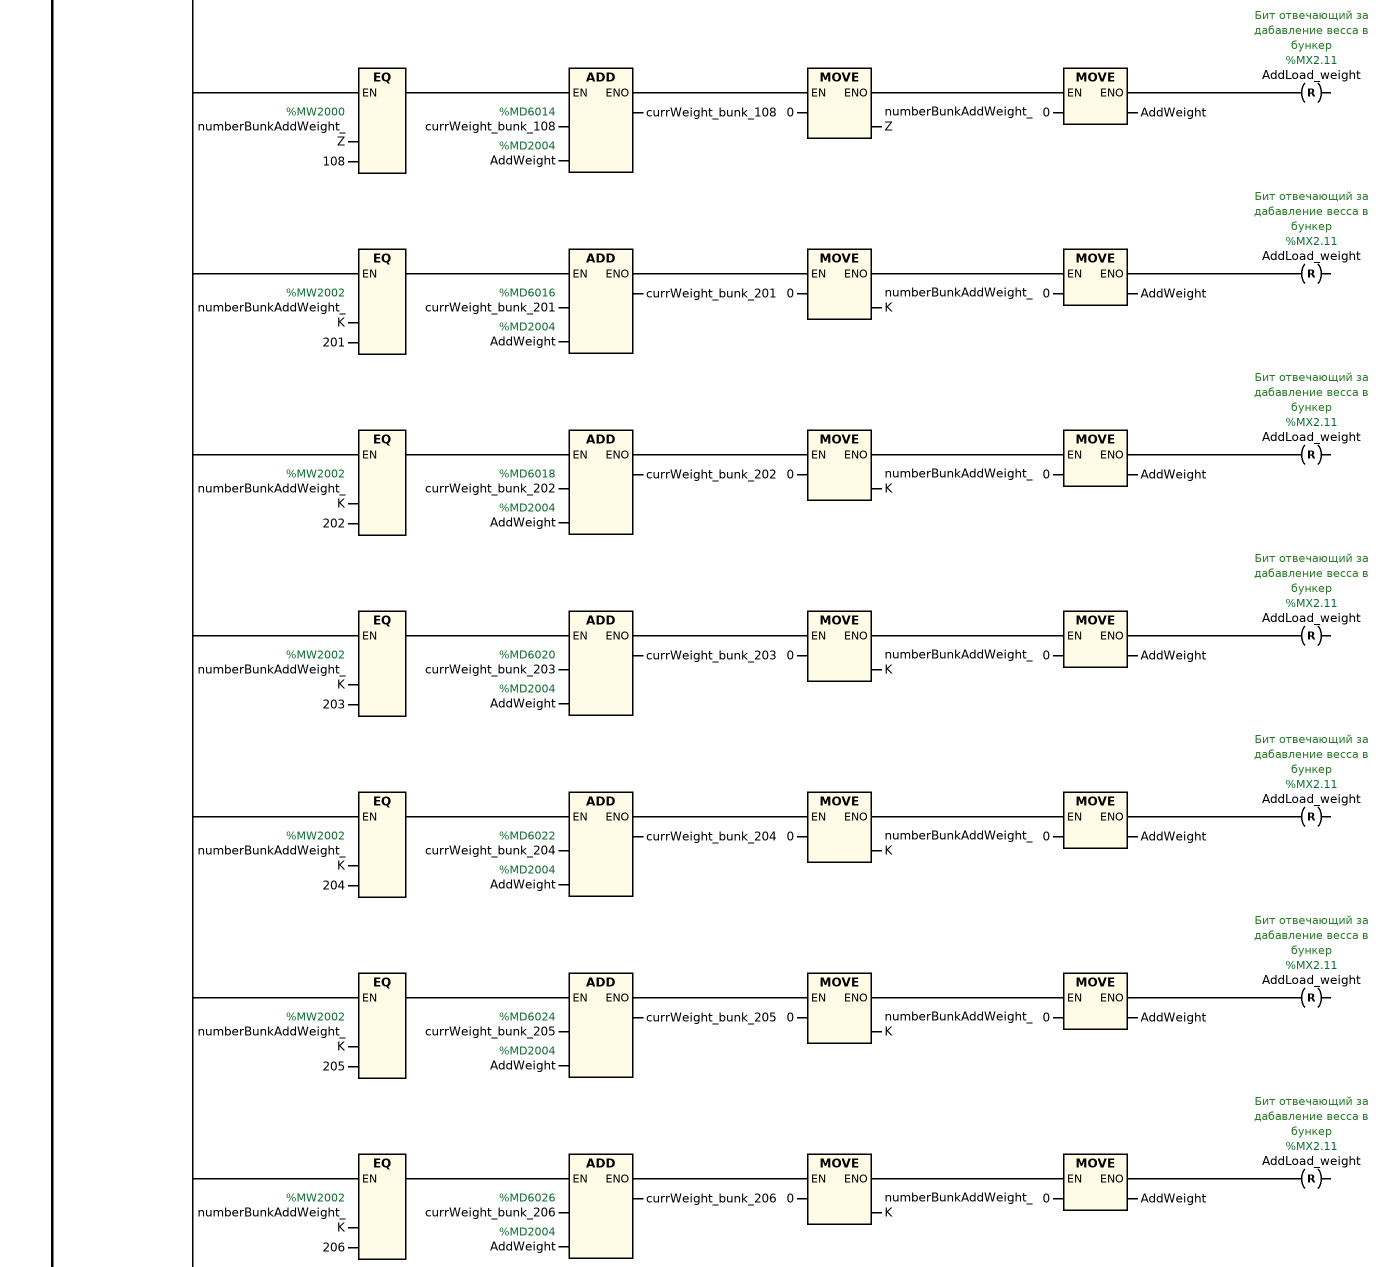
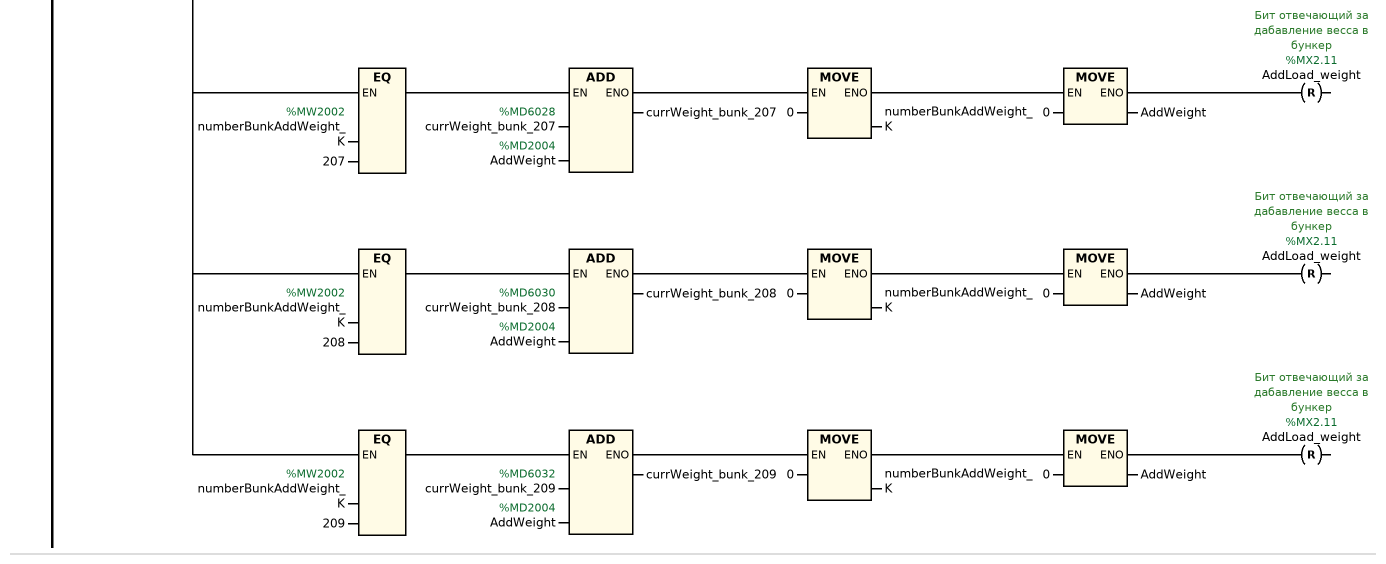
// NETWORK 1
//   AddLoad_weight: Бит отвечающий за дабавление весса в бункер | AT %MX2.11
//   numberBunkAddWeight_Z: Храниться номер бункера для дабавления или удаления значения текущего весса в ручную... Сырье | AT %MW2000
//   currWeight_bunk_101: ----------------------------------------------------------------------------------------------------- текущий вес в зерновых бункерах ----------------------------------------------------------------------------------------------------- | AT %MD6000
//   AddWeight: Значение дабавляемого весса в бункер | AT %MD2004
//   currWeight_bunk_102: AT %MD6002
//   currWeight_bunk_103: AT %MD6004
//   currWeight_bunk_104: AT %MD6006
//   currWeight_bunk_105: AT %MD6008
//   currWeight_bunk_106: AT %MD6010
//   currWeight_bunk_107: AT %MD6012
//   currWeight_bunk_108: AT %MD6014
//   numberBunkAddWeight_K: Храниться номер бункера для дабавления или удаления значения текущего весса в ручную... Добавки | AT %MW2002
//   currWeight_bunk_201: ----------------------------------------------------------------------------------------------------- ----------------------------------------------------------------------------------------------------- текущий вес в бункерах компонентов ----------------------------------------------------------------------------------------------------- | AT %MD6016
//   currWeight_bunk_202: AT %MD6018
//   currWeight_bunk_203: AT %MD6020
//   currWeight_bunk_204: AT %MD6022
//   currWeight_bunk_205: AT %MD6024
//   currWeight_bunk_206: AT %MD6026
//   currWeight_bunk_207: AT %MD6028
//   currWeight_bunk_208: AT %MD6030
//   currWeight_bunk_209: AT %MD6032
_w1 := AddLoad_weight;
IF _w1 AND numberBunkAddWeight_Z = 101 THEN currWeight_bunk_101 := currWeight_bunk_101 + AddWeight; END_IF
IF _w1 AND numberBunkAddWeight_Z = 101 THEN numberBunkAddWeight_Z := 0; END_IF
IF _w1 AND numberBunkAddWeight_Z = 101 THEN AddWeight := 0; END_IF
AddLoad_weight R= _w1 AND numberBunkAddWeight_Z = 101;
IF _w1 AND numberBunkAddWeight_Z = 102 THEN currWeight_bunk_102 := currWeight_bunk_102 + AddWeight; END_IF
IF _w1 AND numberBunkAddWeight_Z = 102 THEN numberBunkAddWeight_Z := 0; END_IF
IF _w1 AND numberBunkAddWeight_Z = 102 THEN AddWeight := 0; END_IF
AddLoad_weight R= _w1 AND numberBunkAddWeight_Z = 102;
IF _w1 AND numberBunkAddWeight_Z = 103 THEN currWeight_bunk_103 := currWeight_bunk_103 + AddWeight; END_IF
IF _w1 AND numberBunkAddWeight_Z = 103 THEN numberBunkAddWeight_Z := 0; END_IF
IF _w1 AND numberBunkAddWeight_Z = 103 THEN AddWeight := 0; END_IF
AddLoad_weight R= _w1 AND numberBunkAddWeight_Z = 103;
IF _w1 AND numberBunkAddWeight_Z = 104 THEN currWeight_bunk_104 := currWeight_bunk_104 + AddWeight; END_IF
IF _w1 AND numberBunkAddWeight_Z = 104 THEN numberBunkAddWeight_Z := 0; END_IF
IF _w1 AND numberBunkAddWeight_Z = 104 THEN AddWeight := 0; END_IF
AddLoad_weight R= _w1 AND numberBunkAddWeight_Z = 104;
IF _w1 AND numberBunkAddWeight_Z = 105 THEN currWeight_bunk_105 := currWeight_bunk_105 + AddWeight; END_IF
IF _w1 AND numberBunkAddWeight_Z = 105 THEN numberBunkAddWeight_Z := 0; END_IF
IF _w1 AND numberBunkAddWeight_Z = 105 THEN AddWeight := 0; END_IF
AddLoad_weight R= _w1 AND numberBunkAddWeight_Z = 105;
IF _w1 AND numberBunkAddWeight_Z = 106 THEN currWeight_bunk_106 := currWeight_bunk_106 + AddWeight; END_IF
IF _w1 AND numberBunkAddWeight_Z = 106 THEN numberBunkAddWeight_Z := 0; END_IF
IF _w1 AND numberBunkAddWeight_Z = 106 THEN AddWeight := 0; END_IF
AddLoad_weight R= _w1 AND numberBunkAddWeight_Z = 106;
IF _w1 AND numberBunkAddWeight_Z = 107 THEN currWeight_bunk_107 := currWeight_bunk_107 + AddWeight; END_IF
IF _w1 AND numberBunkAddWeight_Z = 107 THEN numberBunkAddWeight_Z := 0; END_IF
IF _w1 AND numberBunkAddWeight_Z = 107 THEN AddWeight := 0; END_IF
AddLoad_weight R= _w1 AND numberBunkAddWeight_Z = 107;
IF _w1 AND numberBunkAddWeight_Z = 108 THEN currWeight_bunk_108 := currWeight_bunk_108 + AddWeight; END_IF
IF _w1 AND numberBunkAddWeight_Z = 108 THEN numberBunkAddWeight_Z := 0; END_IF
IF _w1 AND numberBunkAddWeight_Z = 108 THEN AddWeight := 0; END_IF
AddLoad_weight R= _w1 AND numberBunkAddWeight_Z = 108;
IF _w1 AND numberBunkAddWeight_K = 201 THEN currWeight_bunk_201 := currWeight_bunk_201 + AddWeight; END_IF
IF _w1 AND numberBunkAddWeight_K = 201 THEN numberBunkAddWeight_K := 0; END_IF
IF _w1 AND numberBunkAddWeight_K = 201 THEN AddWeight := 0; END_IF
AddLoad_weight R= _w1 AND numberBunkAddWeight_K = 201;
IF _w1 AND numberBunkAddWeight_K = 202 THEN currWeight_bunk_202 := currWeight_bunk_202 + AddWeight; END_IF
IF _w1 AND numberBunkAddWeight_K = 202 THEN numberBunkAddWeight_K := 0; END_IF
IF _w1 AND numberBunkAddWeight_K = 202 THEN AddWeight := 0; END_IF
AddLoad_weight R= _w1 AND numberBunkAddWeight_K = 202;
IF _w1 AND numberBunkAddWeight_K = 203 THEN currWeight_bunk_203 := currWeight_bunk_203 + AddWeight; END_IF
IF _w1 AND numberBunkAddWeight_K = 203 THEN numberBunkAddWeight_K := 0; END_IF
IF _w1 AND numberBunkAddWeight_K = 203 THEN AddWeight := 0; END_IF
AddLoad_weight R= _w1 AND numberBunkAddWeight_K = 203;
IF _w1 AND numberBunkAddWeight_K = 204 THEN currWeight_bunk_204 := currWeight_bunk_204 + AddWeight; END_IF
IF _w1 AND numberBunkAddWeight_K = 204 THEN numberBunkAddWeight_K := 0; END_IF
IF _w1 AND numberBunkAddWeight_K = 204 THEN AddWeight := 0; END_IF
AddLoad_weight R= _w1 AND numberBunkAddWeight_K = 204;
IF _w1 AND numberBunkAddWeight_K = 205 THEN currWeight_bunk_205 := currWeight_bunk_205 + AddWeight; END_IF
IF _w1 AND numberBunkAddWeight_K = 205 THEN numberBunkAddWeight_K := 0; END_IF
IF _w1 AND numberBunkAddWeight_K = 205 THEN AddWeight := 0; END_IF
AddLoad_weight R= _w1 AND numberBunkAddWeight_K = 205;
IF _w1 AND numberBunkAddWeight_K = 206 THEN currWeight_bunk_206 := currWeight_bunk_206 + AddWeight; END_IF
IF _w1 AND numberBunkAddWeight_K = 206 THEN numberBunkAddWeight_K := 0; END_IF
IF _w1 AND numberBunkAddWeight_K = 206 THEN AddWeight := 0; END_IF
AddLoad_weight R= _w1 AND numberBunkAddWeight_K = 206;
IF _w1 AND numberBunkAddWeight_K = 207 THEN currWeight_bunk_207 := currWeight_bunk_207 + AddWeight; END_IF
IF _w1 AND numberBunkAddWeight_K = 207 THEN numberBunkAddWeight_K := 0; END_IF
IF _w1 AND numberBunkAddWeight_K = 207 THEN AddWeight := 0; END_IF
AddLoad_weight R= _w1 AND numberBunkAddWeight_K = 207;
IF _w1 AND numberBunkAddWeight_K = 208 THEN currWeight_bunk_208 := currWeight_bunk_208 + AddWeight; END_IF
IF _w1 AND numberBunkAddWeight_K = 208 THEN numberBunkAddWeight_K := 0; END_IF
IF _w1 AND numberBunkAddWeight_K = 208 THEN AddWeight := 0; END_IF
AddLoad_weight R= _w1 AND numberBunkAddWeight_K = 208;
IF _w1 AND numberBunkAddWeight_K = 209 THEN currWeight_bunk_209 := currWeight_bunk_209 + AddWeight; END_IF
IF _w1 AND numberBunkAddWeight_K = 209 THEN numberBunkAddWeight_K := 0; END_IF
IF _w1 AND numberBunkAddWeight_K = 209 THEN AddWeight := 0; END_IF
AddLoad_weight R= _w1 AND numberBunkAddWeight_K = 209;

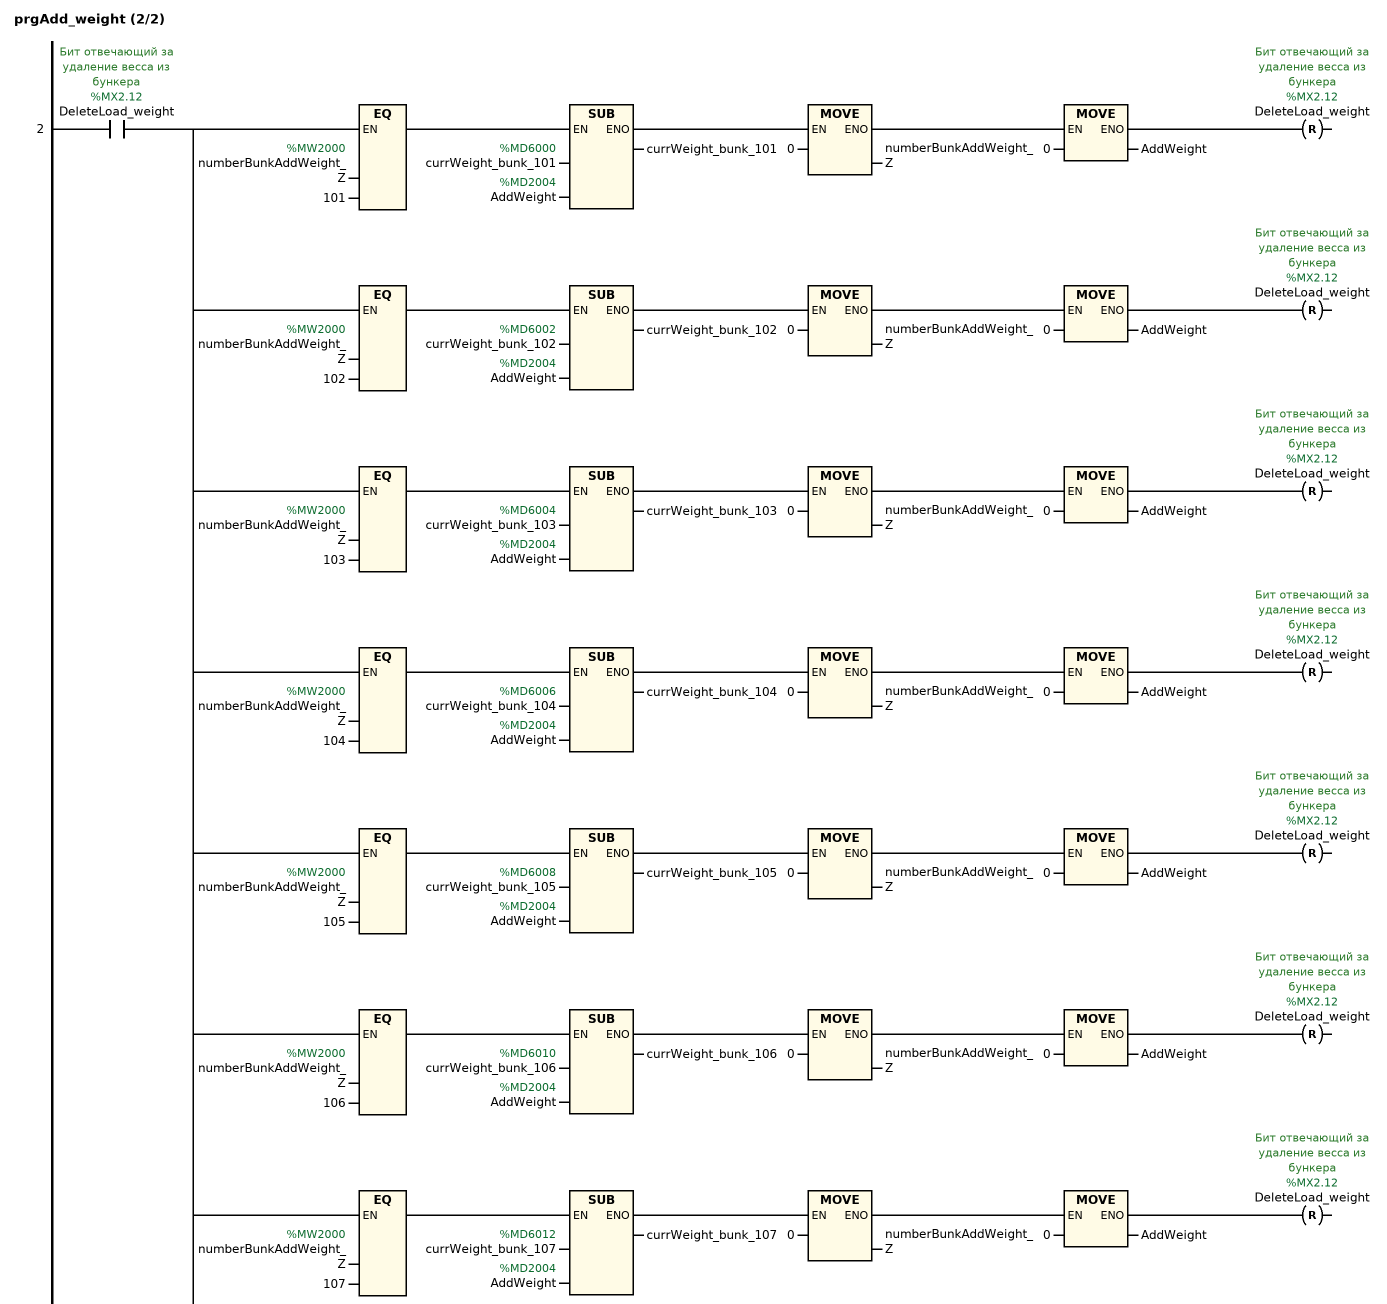
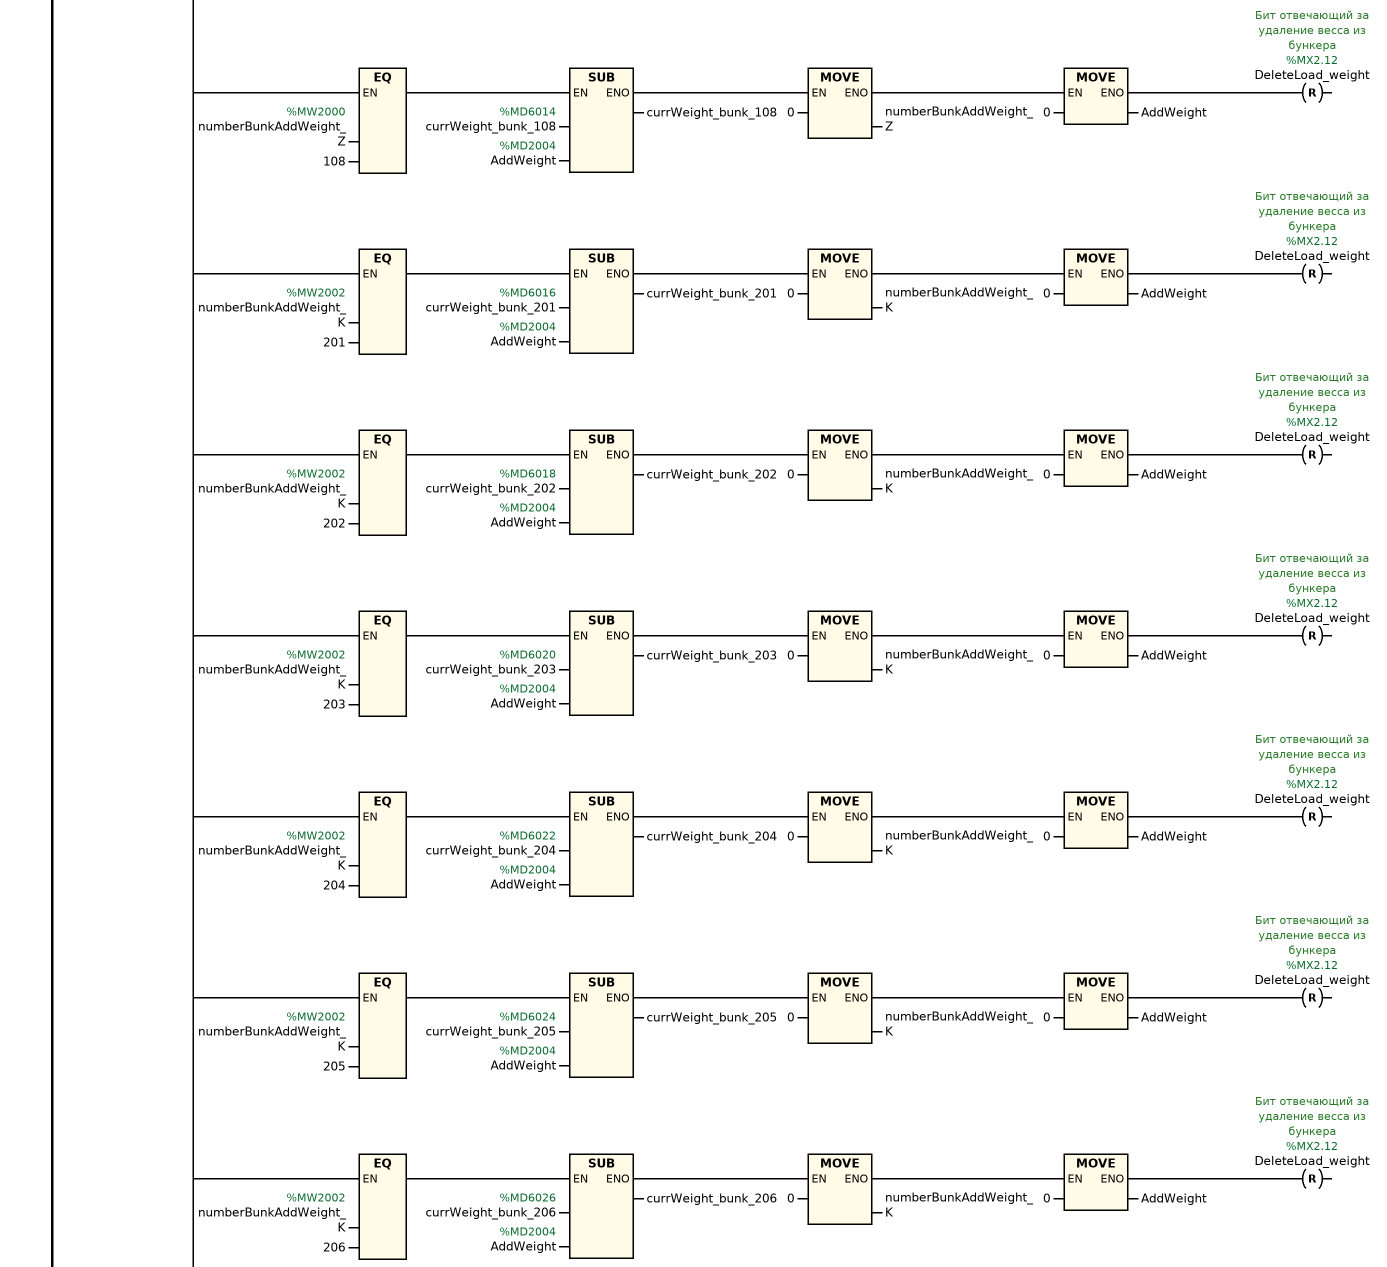
